LIN {X 0,Y 451.554,Z 691.44,A -85,B 0,C 180,E1 7559.051,E2 7559.051} C_VEL
LIN {X 0,Y 450.796,Z 691.44,A -85,B 0,C 180,E1 7568.723,E2 7568.723} C_VEL
LIN {X 0,Y 450.961,Z 693.251,A -85,B 0,C 180,E1 7574.379,E2 7574.379} C_VEL
LIN {X 0,Y 480.104,Z 749.238,A -85,B 0,C 180,E1 7579.793,E2 7579.793} C_VEL
LIN {X 0,Y 479.486,Z 776.375,A -85,B 0,C 180,E1 7581.127,E2 7581.127} C_VEL
LIN {X 0,Y 471.535,Z 837.542,A -85,B 0,C 180,E1 7585.056,E2 7585.056} C_VEL
LIN {X 0,Y 462.67,Z 892.765,A -85,B 0,C 180,E1 7590.85,E2 7590.85} C_VEL
LIN {X 0,Y 455.796,Z 938.399,A -85,B 0,C 180,E1 7598.248,E2 7598.248} C_VEL
LIN {X 0,Y 452.189,Z 968.248,A -85,B 0,C 180,E1 7605.749,E2 7605.749} C_VEL
LIN {X 0,Y 451.04,Z 986.112,A -85,B 0,C 180,E1 7613.349,E2 7613.349} C_VEL
LIN {X 0,Y 450.564,Z 992.815,A -85,B 0,C 180,E1 7620.766,E2 7620.766} C_VEL
LIN {X 0,Y 451.262,Z 989.016,A -85,B 0,C 180,E1 7628.483,E2 7628.483} C_VEL
LIN {X 0,Y 452.265,Z 972.099,A -85,B 0,C 180,E1 7636.86,E2 7636.86} C_VEL
LIN {X 0,Y 455.576,Z 940.536,A -85,B 0,C 180,E1 7645.223,E2 7645.223} C_VEL
LIN {X 0,Y 462.458,Z 894.509,A -85,B 0,C 180,E1 7652.822,E2 7652.822} C_VEL
LIN {X 0,Y 471.275,Z 839.468,A -85,B 0,C 180,E1 7658.682,E2 7658.682} C_VEL
LIN {X 0,Y 479.234,Z 777.254,A -85,B 0,C 180,E1 7662.749,E2 7662.749} C_VEL
LIN {X 0,Y 480.534,Z 748.867,A -85,B 0,C 180,E1 7664.089,E2 7664.089} C_VEL
LIN {X 0,Y 451.925,Z 695.998,A -85,B 0,C 180,E1 7669.283,E2 7669.283} C_VEL
LIN {X 0,Y 450.465,Z 691.44,A -85,B 0,C 180,E1 7669.758,E2 7669.758} C_VEL
LIN {X 0,Y 450.136,Z 691.44,A -85,B 0,C 180,E1 7679.266,E2 7679.266} C_VEL
LIN {X 0,Y 449.936,Z 691.44,A -85,B 0,C 180,E1 7688.608,E2 7688.608} C_VEL
LIN {X 0,Y 449.949,Z 691.44,A -85,B 0,C 180,E1 7698.876,E2 7698.876} C_VEL
LIN {X 0,Y 450.069,Z 691.44,A -85,B 0,C 180,E1 7709.299,E2 7709.299} C_VEL
LIN {X 0,Y 449.954,Z 691.44,A -85,B 0,C 180,E1 7719.253,E2 7719.253} C_VEL
LIN {X 0,Y 450.985,Z 691.44,A -85,B 0,C 180,E1 7727.357,E2 7727.357} C_VEL
LIN {X 0,Y 450.837,Z 691.44,A -85,B 0,C 180,E1 7737.094,E2 7737.094} C_VEL
LIN {X 0,Y 450.806,Z 691.44,A -85,B 0,C 180,E1 7744.813,E2 7744.813} C_VEL
LIN {X 0,Y 450.666,Z 691.44,A -85,B 0,C 180,E1 7754.61,E2 7754.61} C_VEL
LIN {X 0,Y 450.257,Z 691.44,A -85,B 0,C 180,E1 7764.893,E2 7764.893} C_VEL
LIN {X 0,Y 449.84,Z 691.44,A -85,B 0,C 180,E1 7774.255,E2 7774.255} C_VEL
LIN {X 0,Y 450.159,Z 693.285,A -85,B 0,C 180,E1 7781.816,E2 7781.816} C_VEL
LIN {X 0,Y 483.227,Z 752.373,A -85,B 0,C 180,E1 7787.254,E2 7787.254} C_VEL
LIN {X 0,Y 477.78,Z 816.561,A -85,B 0,C 180,E1 7789.78,E2 7789.78} C_VEL
LIN {X 0,Y 469.391,Z 878.673,A -85,B 0,C 180,E1 7794.175,E2 7794.175} C_VEL
LIN {X 0,Y 468.305,Z 886.117,A -85,B 0,C 180,E1 7794.87,E2 7794.87} C_VEL
LIN {X 0,Y 457.031,Z 913.56,A -85,B 0,C 180,E1 7797.288,E2 7797.288} C_VEL
LIN {X 0,Y 449.955,Z 959.158,A -85,B 0,C 180,E1 7804.083,E2 7804.083} C_VEL
LIN {X 0,Y 445.282,Z 994.231,A -85,B 0,C 180,E1 7812.256,E2 7812.256} C_VEL
LIN {X 0,Y 443.447,Z 1014.285,A -85,B 0,C 180,E1 7820.147,E2 7820.147} C_VEL
LIN {X 0,Y 443.05,Z 1022.147,A -85,B 0,C 180,E1 7827.054,E2 7827.054} C_VEL
LIN {X 0,Y 443.063,Z 1020.767,A -85,B 0,C 180,E1 7834.912,E2 7834.912} C_VEL
LIN {X 0,Y 443.75,Z 1007.555,A -85,B 0,C 180,E1 7843.07,E2 7843.07} C_VEL
LIN {X 0,Y 447.084,Z 979.442,A -85,B 0,C 180,E1 7851.662,E2 7851.662} C_VEL
LIN {X 0,Y 453.089,Z 938.558,A -85,B 0,C 180,E1 7859.353,E2 7859.353} C_VEL
LIN {X 0,Y 461.64,Z 883.668,A -85,B 0,C 180,E1 7865.91,E2 7865.91} C_VEL
LIN {X 0,Y 470.623,Z 820.966,A -85,B 0,C 180,E1 7870.566,E2 7870.566} C_VEL
LIN {X 0,Y 476.046,Z 752.177,A -85,B 0,C 180,E1 7873.483,E2 7873.483} C_VEL
LIN {X 0,Y 441.94,Z 691.44,A -85,B 0,C 180,E1 7879.572,E2 7879.572} C_VEL
LIN {X 0,Y 442.027,Z 691.44,A -85,B 0,C 180,E1 7890.171,E2 7890.171} C_VEL
LIN {X 0,Y 442.1,Z 691.44,A -85,B 0,C 180,E1 7900.989,E2 7900.989} C_VEL
LIN {X 0,Y 442.87,Z 691.44,A -85,B 0,C 180,E1 7911.146,E2 7911.146} C_VEL
LIN {X 0,Y 443.032,Z 691.44,A -85,B 0,C 180,E1 7920.994,E2 7920.994} C_VEL
LIN {X 0,Y 442.705,Z 691.44,A -85,B 0,C 180,E1 7930.877,E2 7930.877} C_VEL
LIN {X 0,Y 442.98,Z 693.318,A -85,B 0,C 180,E1 7933.215,E2 7933.215} C_VEL
LIN {X 0,Y 472.547,Z 748.959,A -85,B 0,C 180,E1 7938.943,E2 7938.943} C_VEL
LIN {X 0,Y 474.866,Z 762.006,A -85,B 0,C 180,E1 7939.835,E2 7939.835} C_VEL
LIN {X 0,Y 466.818,Z 825.923,A -85,B 0,C 180,E1 7943.512,E2 7943.512} C_VEL
LIN {X 0,Y 457.64,Z 882.015,A -85,B 0,C 180,E1 7948.928,E2 7948.928} C_VEL
LIN {X 0,Y 449.947,Z 928.738,A -85,B 0,C 180,E1 7955.962,E2 7955.962} C_VEL
LIN {X 0,Y 445.038,Z 964.744,A -85,B 0,C 180,E1 7964.35,E2 7964.35} C_VEL
LIN {X 0,Y 443.257,Z 984.655,A -85,B 0,C 180,E1 7972.336,E2 7972.336} C_VEL
LIN {X 0,Y 442.582,Z 992.719,A -85,B 0,C 180,E1 7980.186,E2 7980.186} C_VEL
LIN {X 0,Y 443.266,Z 988.627,A -85,B 0,C 180,E1 7988.932,E2 7988.932} C_VEL
LIN {X 0,Y 444.309,Z 970.625,A -85,B 0,C 180,E1 7997.674,E2 7997.674} C_VEL
LIN {X 0,Y 447.986,Z 939.674,A -85,B 0,C 180,E1 8005.832,E2 8005.832} C_VEL
LIN {X 0,Y 455.506,Z 893.468,A -85,B 0,C 180,E1 8013.528,E2 8013.528} C_VEL
LIN {X 0,Y 464.916,Z 838.34,A -85,B 0,C 180,E1 8019.394,E2 8019.394} C_VEL
LIN {X 0,Y 473.409,Z 775.784,A -85,B 0,C 180,E1 8023.457,E2 8023.457} C_VEL
LIN {X 0,Y 474.106,Z 751.685,A -85,B 0,C 180,E1 8024.661,E2 8024.661} C_VEL
LIN {X 0,Y 445.382,Z 697.645,A -85,B 0,C 180,E1 8030.143,E2 8030.143} C_VEL
LIN {X 0,Y 442.399,Z 691.44,A -85,B 0,C 180,E1 8031.112,E2 8031.112} C_VEL
LIN {X 0,Y 442.119,Z 691.44,A -85,B 0,C 180,E1 8039.85,E2 8039.85} C_VEL
LIN {X 0,Y 441.891,Z 691.44,A -85,B 0,C 180,E1 8049.446,E2 8049.446} C_VEL
LIN {X 0,Y 441.873,Z 691.44,A -85,B 0,C 180,E1 8057.955,E2 8057.955} C_VEL
LIN {X 0,Y 441.946,Z 691.44,A -85,B 0,C 180,E1 8067.839,E2 8067.839} C_VEL
LIN {X 0,Y 441.935,Z 691.44,A -85,B 0,C 180,E1 8076.734,E2 8076.734} C_VEL
LIN {X 0,Y 442.969,Z 691.44,A -85,B 0,C 180,E1 8087.528,E2 8087.528} C_VEL
LIN {X 0,Y 442.866,Z 691.44,A -85,B 0,C 180,E1 8097.041,E2 8097.041} C_VEL
LIN {X 0,Y 442.821,Z 691.44,A -85,B 0,C 180,E1 8104.9,E2 8104.9} C_VEL
LIN {X 0,Y 442.657,Z 691.44,A -85,B 0,C 180,E1 8114.88,E2 8114.88} C_VEL
LIN {X 0,Y 442.205,Z 691.44,A -85,B 0,C 180,E1 8125.379,E2 8125.379} C_VEL
LIN {X 0,Y 441.848,Z 691.44,A -85,B 0,C 180,E1 8136.182,E2 8136.182} C_VEL
LIN {X 0,Y 442.043,Z 692.748,A -85,B 0,C 180,E1 8140.669,E2 8140.669} C_VEL
LIN {X 0,Y 477.063,Z 755.273,A -85,B 0,C 180,E1 8146.678,E2 8146.678} C_VEL
LIN {X 0,Y 471.042,Z 819.946,A -85,B 0,C 180,E1 8149.353,E2 8149.353} C_VEL
LIN {X 0,Y 462.246,Z 881.197,A -85,B 0,C 180,E1 8153.834,E2 8153.834} C_VEL
LIN {X 0,Y 457.031,Z 913.56,A -85,B 0,C 180,E1 8157.288,E2 8157.288} C_VEL
LIN {X 0,Y 445.432,Z 938.523,A -85,B 0,C 180,E1 8160.14,E2 8160.14} C_VEL
LIN {X 0,Y 438.964,Z 978.353,A -85,B 0,C 180,E1 8167.648,E2 8167.648} C_VEL
LIN {X 0,Y 435.816,Z 1004.336,A -85,B 0,C 180,E1 8175.377,E2 8175.377} C_VEL
LIN {X 0,Y 435.092,Z 1019.244,A -85,B 0,C 180,E1 8183.454,E2 8183.454} C_VEL
LIN {X 0,Y 435.342,Z 1022.837,A -85,B 0,C 180,E1 8190.998,E2 8190.998} C_VEL
LIN {X 0,Y 435.357,Z 1015.886,A -85,B 0,C 180,E1 8199.024,E2 8199.024} C_VEL
LIN {X 0,Y 436.862,Z 995.719,A -85,B 0,C 180,E1 8207.643,E2 8207.643} C_VEL
LIN {X 0,Y 441.422,Z 962.929,A -85,B 0,C 180,E1 8215.664,E2 8215.664} C_VEL
LIN {X 0,Y 449.432,Z 915.459,A -85,B 0,C 180,E1 8222.997,E2 8222.997} C_VEL
LIN {X 0,Y 459.298,Z 857.062,A -85,B 0,C 180,E1 8228.768,E2 8228.768} C_VEL
LIN {X 0,Y 467.582,Z 794.293,A -85,B 0,C 180,E1 8232.533,E2 8232.533} C_VEL
LIN {X 0,Y 469.791,Z 755.185,A -85,B 0,C 180,E1 8234.086,E2 8234.086} C_VEL
LIN {X 0,Y 436.487,Z 697.36,A -85,B 0,C 180,E1 8240.149,E2 8240.149} C_VEL
LIN {X 0,Y 433.802,Z 691.44,A -85,B 0,C 180,E1 8240.877,E2 8240.877} C_VEL
LIN {X 0,Y 434.008,Z 691.44,A -85,B 0,C 180,E1 8251.859,E2 8251.859} C_VEL
LIN {X 0,Y 434.256,Z 691.44,A -85,B 0,C 180,E1 8262.74,E2 8262.74} C_VEL
LIN {X 0,Y 434.924,Z 691.44,A -85,B 0,C 180,E1 8273.001,E2 8273.001} C_VEL
LIN {X 0,Y 435.026,Z 691.44,A -85,B 0,C 180,E1 8281.013,E2 8281.013} C_VEL
LIN {X 0,Y 434.694,Z 691.44,A -85,B 0,C 180,E1 8291.08,E2 8291.08} C_VEL
LIN {X 0,Y 435.021,Z 693.636,A -85,B 0,C 180,E1 8291.977,E2 8291.977} C_VEL
LIN {X 0,Y 464.673,Z 747.641,A -85,B 0,C 180,E1 8297.959,E2 8297.959} C_VEL
LIN {X 0,Y 468.849,Z 762.644,A -85,B 0,C 180,E1 8299.199,E2 8299.199} C_VEL
LIN {X 0,Y 460.363,Z 826.705,A -85,B 0,C 180,E1 8302.927,E2 8302.927} C_VEL
LIN {X 0,Y 450.621,Z 882.973,A -85,B 0,C 180,E1 8308.447,E2 8308.447} C_VEL
LIN {X 0,Y 442.51,Z 928.888,A -85,B 0,C 180,E1 8315.491,E2 8315.491} C_VEL
LIN {X 0,Y 437.286,Z 964.581,A -85,B 0,C 180,E1 8323.978,E2 8323.978} C_VEL
LIN {X 0,Y 435.243,Z 985.065,A -85,B 0,C 180,E1 8332.398,E2 8332.398} C_VEL
LIN {X 0,Y 434.561,Z 992.463,A -85,B 0,C 180,E1 8339.578,E2 8339.578} C_VEL
LIN {X 0,Y 435.121,Z 990.295,A -85,B 0,C 180,E1 8347.542,E2 8347.542} C_VEL
LIN {X 0,Y 436.37,Z 974.559,A -85,B 0,C 180,E1 8356.49,E2 8356.49} C_VEL
LIN {X 0,Y 439.717,Z 945.125,A -85,B 0,C 180,E1 8365.051,E2 8365.051} C_VEL
LIN {X 0,Y 447.115,Z 901.895,A -85,B 0,C 180,E1 8372.919,E2 8372.919} C_VEL
LIN {X 0,Y 456.677,Z 848.952,A -85,B 0,C 180,E1 8379.082,E2 8379.082} C_VEL
LIN {X 0,Y 465.74,Z 787.5,A -85,B 0,C 180,E1 8383.545,E2 8383.545} C_VEL
LIN {X 0,Y 468.049,Z 755.229,A -85,B 0,C 180,E1 8385.176,E2 8385.176} C_VEL
LIN {X 0,Y 440.965,Z 703.44,A -85,B 0,C 180,E1 8390.624,E2 8390.624} C_VEL
LIN {X 0,Y 434.298,Z 691.44,A -85,B 0,C 180,E1 8392.194,E2 8392.194} C_VEL
LIN {X 0,Y 433.924,Z 691.44,A -85,B 0,C 180,E1 8402.827,E2 8402.827} C_VEL
LIN {X 0,Y 433.83,Z 691.44,A -85,B 0,C 180,E1 8413.011,E2 8413.011} C_VEL
LIN {X 0,Y 433.75,Z 691.44,A -85,B 0,C 180,E1 8422.244,E2 8422.244} C_VEL
LIN {X 0,Y 434.015,Z 691.44,A -85,B 0,C 180,E1 8433.081,E2 8433.081} C_VEL
LIN {X 0,Y 434.843,Z 691.44,A -85,B 0,C 180,E1 8444.818,E2 8444.818} C_VEL
LIN {X 0,Y 435.01,Z 691.44,A -85,B 0,C 180,E1 8454.985,E2 8454.985} C_VEL
LIN {X 0,Y 435.081,Z 691.44,A -85,B 0,C 180,E1 8462.984,E2 8462.984} C_VEL
LIN {X 0,Y 434.639,Z 691.44,A -85,B 0,C 180,E1 8473.099,E2 8473.099} C_VEL
LIN {X 0,Y 434.257,Z 691.44,A -85,B 0,C 180,E1 8483.672,E2 8483.672} C_VEL
LIN {X 0,Y 433.815,Z 691.44,A -85,B 0,C 180,E1 8494.705,E2 8494.705} C_VEL
LIN {X 0,Y 433.956,Z 692.746,A -85,B 0,C 180,E1 8499.468,E2 8499.468} C_VEL
LIN {X 0,Y 469.825,Z 755.777,A -85,B 0,C 180,E1 8505.884,E2 8505.884} C_VEL
LIN {X 0,Y 464.026,Z 825.724,A -85,B 0,C 180,E1 8509.052,E2 8509.052} C_VEL
LIN {X 0,Y 454.868,Z 884.496,A -85,B 0,C 180,E1 8513.572,E2 8513.572} C_VEL
LIN {X 0,Y 445.432,Z 938.523,A -85,B 0,C 180,E1 8520.14,E2 8520.14} C_VEL
LIN {X 0,Y 434.61,Z 960.552,A -85,B 0,C 180,E1 8523.479,E2 8523.479} C_VEL
LIN {X 0,Y 429.713,Z 993.824,A -85,B 0,C 180,E1 8531.467,E2 8531.467} C_VEL
LIN {X 0,Y 427.573,Z 1014.285,A -85,B 0,C 180,E1 8539.777,E2 8539.777} C_VEL
LIN {X 0,Y 427.056,Z 1022.147,A -85,B 0,C 180,E1 8546.944,E2 8546.944} C_VEL
LIN {X 0,Y 427.087,Z 1020.766,A -85,B 0,C 180,E1 8555.096,E2 8555.096} C_VEL
LIN {X 0,Y 428.068,Z 1006.921,A -85,B 0,C 180,E1 8563.845,E2 8563.845} C_VEL
LIN {X 0,Y 431.896,Z 978.302,A -85,B 0,C 180,E1 8572.737,E2 8572.737} C_VEL
LIN {X 0,Y 438.853,Z 936.044,A -85,B 0,C 180,E1 8580.668,E2 8580.668} C_VEL
LIN {X 0,Y 448.501,Z 881.198,A -85,B 0,C 180,E1 8587.31,E2 8587.31} C_VEL
LIN {X 0,Y 458.407,Z 817.94,A -85,B 0,C 180,E1 8592.02,E2 8592.02} C_VEL
LIN {X 0,Y 463.715,Z 758.59,A -85,B 0,C 180,E1 8594.657,E2 8594.657} C_VEL
LIN {X 0,Y 432.524,Z 703.466,A -85,B 0,C 180,E1 8600.626,E2 8600.626} C_VEL
LIN {X 0,Y 425.74,Z 691.44,A -85,B 0,C 180,E1 8602.433,E2 8602.433} C_VEL
LIN {X 0,Y 425.979,Z 691.44,A -85,B 0,C 180,E1 8613.582,E2 8613.582} C_VEL
LIN {X 0,Y 426.337,Z 691.44,A -85,B 0,C 180,E1 8624.536,E2 8624.536} C_VEL
LIN {X 0,Y 426.827,Z 691.44,A -85,B 0,C 180,E1 8634.916,E2 8634.916} C_VEL
LIN {X 0,Y 426.878,Z 691.44,A -85,B 0,C 180,E1 8643.07,E2 8643.07} C_VEL
LIN {X 0,Y 426.829,Z 693.053,A -85,B 0,C 180,E1 8650.574,E2 8650.574} C_VEL
LIN {X 0,Y 456.913,Z 746.746,A -85,B 0,C 180,E1 8656.957,E2 8656.957} C_VEL
LIN {X 0,Y 462.493,Z 766.687,A -85,B 0,C 180,E1 8658.693,E2 8658.693} C_VEL
LIN {X 0,Y 453.603,Z 829.727,A -85,B 0,C 180,E1 8662.495,E2 8662.495} C_VEL
LIN {X 0,Y 443.125,Z 886.449,A -85,B 0,C 180,E1 8668.262,E2 8668.262} C_VEL
LIN {X 0,Y 434.551,Z 932.151,A -85,B 0,C 180,E1 8675.584,E2 8675.584} C_VEL
LIN {X 0,Y 428.946,Z 967.211,A -85,B 0,C 180,E1 8684.489,E2 8684.489} C_VEL
LIN {X 0,Y 427.137,Z 986.415,A -85,B 0,C 180,E1 8693.07,E2 8693.07} C_VEL
LIN {X 0,Y 426.463,Z 992.905,A -85,B 0,C 180,E1 8701.289,E2 8701.289} C_VEL
LIN {X 0,Y 427.2,Z 988.636,A -85,B 0,C 180,E1 8709.193,E2 8709.193} C_VEL
LIN {X 0,Y 428.407,Z 971.752,A -85,B 0,C 180,E1 8717.843,E2 8717.843} C_VEL
LIN {X 0,Y 432.819,Z 939.838,A -85,B 0,C 180,E1 8726.734,E2 8726.734} C_VEL
LIN {X 0,Y 441.104,Z 895.84,A -85,B 0,C 180,E1 8734.382,E2 8734.382} C_VEL
LIN {X 0,Y 451.537,Z 841.543,A -85,B 0,C 180,E1 8740.408,E2 8740.408} C_VEL
LIN {X 0,Y 461.059,Z 778.462,A -85,B 0,C 180,E1 8744.659,E2 8744.659} C_VEL
LIN {X 0,Y 461.808,Z 758.295,A -85,B 0,C 180,E1 8745.753,E2 8745.753} C_VEL
LIN {X 0,Y 436.098,Z 708.579,A -85,B 0,C 180,E1 8751.184,E2 8751.184} C_VEL
LIN {X 0,Y 426.272,Z 691.44,A -85,B 0,C 180,E1 8753.157,E2 8753.157} C_VEL
LIN {X 0,Y 425.866,Z 691.44,A -85,B 0,C 180,E1 8763.529,E2 8763.529} C_VEL
LIN {X 0,Y 425.806,Z 691.44,A -85,B 0,C 180,E1 8774.027,E2 8774.027} C_VEL
LIN {X 0,Y 425.748,Z 691.44,A -85,B 0,C 180,E1 8783.972,E2 8783.972} C_VEL
LIN {X 0,Y 426.016,Z 691.44,A -85,B 0,C 180,E1 8793.553,E2 8793.553} C_VEL
LIN {X 0,Y 426.78,Z 691.44,A -85,B 0,C 180,E1 8804.524,E2 8804.524} C_VEL
LIN {X 0,Y 427.001,Z 691.44,A -85,B 0,C 180,E1 8814.89,E2 8814.89} C_VEL
LIN {X 0,Y 427.065,Z 691.44,A -85,B 0,C 180,E1 8823.041,E2 8823.041} C_VEL
LIN {X 0,Y 426.619,Z 691.44,A -85,B 0,C 180,E1 8833.35,E2 8833.35} C_VEL
LIN {X 0,Y 426.172,Z 691.44,A -85,B 0,C 180,E1 8844.15,E2 8844.15} C_VEL
LIN {X 0,Y 425.796,Z 691.44,A -85,B 0,C 180,E1 8853.504,E2 8853.504} C_VEL
LIN {X 0,Y 425.926,Z 693.215,A -85,B 0,C 180,E1 8858.227,E2 8858.227} C_VEL
LIN {X 0,Y 461.569,Z 754.086,A -85,B 0,C 180,E1 8864.861,E2 8864.861} C_VEL
LIN {X 0,Y 464.491,Z 766.283,A -85,B 0,C 180,E1 8865.689,E2 8865.689} C_VEL
LIN {X 0,Y 456.915,Z 831.706,A -85,B 0,C 180,E1 8868.774,E2 8868.774} C_VEL
LIN {X 0,Y 446.908,Z 891.589,A -85,B 0,C 180,E1 8873.698,E2 8873.698} C_VEL
LIN {X 0,Y 437.196,Z 943.334,A -85,B 0,C 180,E1 8880.424,E2 8880.424} C_VEL
LIN {X 0,Y 434.61,Z 960.552,A -85,B 0,C 180,E1 8883.479,E2 8883.479} C_VEL
LIN {X 0,Y 423.366,Z 979.613,A -85,B 0,C 180,E1 8887.193,E2 8887.193} C_VEL
LIN {X 0,Y 419.891,Z 1005.675,A -85,B 0,C 180,E1 8895.345,E2 8895.345} C_VEL
LIN {X 0,Y 419.067,Z 1018.682,A -85,B 0,C 180,E1 8902.718,E2 8902.718} C_VEL
LIN {X 0,Y 419.337,Z 1022.836,A -85,B 0,C 180,E1 8911.036,E2 8911.036} C_VEL
LIN {X 0,Y 419.336,Z 1015.886,A -85,B 0,C 180,E1 8919.372,E2 8919.372} C_VEL
LIN {X 0,Y 420.99,Z 997.104,A -85,B 0,C 180,E1 8927.843,E2 8927.843} C_VEL
LIN {X 0,Y 425.962,Z 964.688,A -85,B 0,C 180,E1 8936.132,E2 8936.132} C_VEL
LIN {X 0,Y 434.995,Z 916.695,A -85,B 0,C 180,E1 8943.931,E2 8943.931} C_VEL
LIN {X 0,Y 446.071,Z 858.144,A -85,B 0,C 180,E1 8949.93,E2 8949.93} C_VEL
LIN {X 0,Y 455.377,Z 795.802,A -85,B 0,C 180,E1 8953.801,E2 8953.801} C_VEL
LIN {X 0,Y 457.53,Z 761.525,A -85,B 0,C 180,E1 8955.277,E2 8955.277} C_VEL
LIN {X 0,Y 428.214,Z 708.933,A -85,B 0,C 180,E1 8961.2,E2 8961.2} C_VEL
LIN {X 0,Y 417.729,Z 691.44,A -85,B 0,C 180,E1 8963.636,E2 8963.636} C_VEL
LIN {X 0,Y 417.903,Z 691.44,A -85,B 0,C 180,E1 8973.03,E2 8973.03} C_VEL
LIN {X 0,Y 418.277,Z 691.44,A -85,B 0,C 180,E1 8984.23,E2 8984.23} C_VEL
LIN {X 0,Y 418.828,Z 691.44,A -85,B 0,C 180,E1 8995.16,E2 8995.16} C_VEL
LIN {X 0,Y 418.875,Z 691.44,A -85,B 0,C 180,E1 9003.128,E2 9003.128} C_VEL
LIN {X 0,Y 418.957,Z 693.291,A -85,B 0,C 180,E1 9009.129,E2 9009.129} C_VEL
LIN {X 0,Y 447.481,Z 742.324,A -85,B 0,C 180,E1 9015.519,E2 9015.519} C_VEL
LIN {X 0,Y 456.404,Z 769.016,A -85,B 0,C 180,E1 9018.099,E2 9018.099} C_VEL
LIN {X 0,Y 447.195,Z 830.655,A -85,B 0,C 180,E1 9021.892,E2 9021.892} C_VEL
LIN {X 0,Y 436.217,Z 887.146,A -85,B 0,C 180,E1 9027.722,E2 9027.722} C_VEL
LIN {X 0,Y 427.316,Z 931.762,A -85,B 0,C 180,E1 9034.962,E2 9034.962} C_VEL
LIN {X 0,Y 421.506,Z 965.772,A -85,B 0,C 180,E1 9043.661,E2 9043.661} C_VEL
LIN {X 0,Y 419.279,Z 985.435,A -85,B 0,C 180,E1 9052.258,E2 9052.258} C_VEL
LIN {X 0,Y 418.483,Z 992.818,A -85,B 0,C 180,E1 9060.688,E2 9060.688} C_VEL
LIN {X 0,Y 419.2,Z 989.225,A -85,B 0,C 180,E1 9068.776,E2 9068.776} C_VEL
LIN {X 0,Y 420.446,Z 972.894,A -85,B 0,C 180,E1 9077.704,E2 9077.704} C_VEL
LIN {X 0,Y 424.898,Z 942.401,A -85,B 0,C 180,E1 9086.673,E2 9086.673} C_VEL
LIN {X 0,Y 433.661,Z 898.569,A -85,B 0,C 180,E1 9094.612,E2 9094.612} C_VEL
LIN {X 0,Y 444.87,Z 843.076,A -85,B 0,C 180,E1 9100.939,E2 9100.939} C_VEL
LIN {X 0,Y 454.776,Z 780.809,A -85,B 0,C 180,E1 9105.236,E2 9105.236} C_VEL
LIN {X 0,Y 455.561,Z 761.257,A -85,B 0,C 180,E1 9106.35,E2 9106.35} C_VEL
LIN {X 0,Y 429.428,Z 710.166,A -85,B 0,C 180,E1 9112.142,E2 9112.142} C_VEL
LIN {X 0,Y 418.215,Z 691.44,A -85,B 0,C 180,E1 9114.665,E2 9114.665} C_VEL
LIN {X 0,Y 417.701,Z 691.44,A -85,B 0,C 180,E1 9125.172,E2 9125.172} C_VEL
LIN {X 0,Y 417.747,Z 691.44,A -85,B 0,C 180,E1 9135.105,E2 9135.105} C_VEL
LIN {X 0,Y 417.746,Z 691.44,A -85,B 0,C 180,E1 9145.727,E2 9145.727} C_VEL
LIN {X 0,Y 417.943,Z 691.44,A -85,B 0,C 180,E1 9155.312,E2 9155.312} C_VEL
LIN {X 0,Y 418.876,Z 691.44,A -85,B 0,C 180,E1 9166.37,E2 9166.37} C_VEL
LIN {X 0,Y 418.869,Z 691.44,A -85,B 0,C 180,E1 9176.872,E2 9176.872} C_VEL
LIN {X 0,Y 418.832,Z 691.44,A -85,B 0,C 180,E1 9185.181,E2 9185.181} C_VEL
LIN {X 0,Y 418.489,Z 691.44,A -85,B 0,C 180,E1 9196.056,E2 9196.056} C_VEL
LIN {X 0,Y 418,Z 691.44,A -85,B 0,C 180,E1 9207.189,E2 9207.189} C_VEL
LIN {X 0,Y 417.818,Z 692.822,A -85,B 0,C 180,E1 9216.873,E2 9216.873} C_VEL
LIN {X 0,Y 454.81,Z 755.444,A -85,B 0,C 180,E1 9224.079,E2 9224.079} C_VEL
LIN {X 0,Y 458.441,Z 768.769,A -85,B 0,C 180,E1 9225.079,E2 9225.079} C_VEL
LIN {X 0,Y 450.44,Z 833.237,A -85,B 0,C 180,E1 9228.216,E2 9228.216} C_VEL
LIN {X 0,Y 439.853,Z 893.141,A -85,B 0,C 180,E1 9233.253,E2 9233.253} C_VEL
LIN {X 0,Y 429.326,Z 946.123,A -85,B 0,C 180,E1 9240.387,E2 9240.387} C_VEL
LIN {X 0,Y 423.366,Z 979.613,A -85,B 0,C 180,E1 9247.193,E2 9247.193} C_VEL
LIN {X 0,Y 413.778,Z 995.457,A -85,B 0,C 180,E1 9251.347,E2 9251.347} C_VEL
LIN {X 0,Y 411.346,Z 1015.885,A -85,B 0,C 180,E1 9260.443,E2 9260.443} C_VEL
LIN {X 0,Y 410.914,Z 1022.836,A -85,B 0,C 180,E1 9268.941,E2 9268.941} C_VEL
LIN {X 0,Y 411.395,Z 1018.684,A -85,B 0,C 180,E1 9277.418,E2 9277.418} C_VEL
LIN {X 0,Y 412.834,Z 1001.069,A -85,B 0,C 180,E1 9286.72,E2 9286.72} C_VEL
LIN {X 0,Y 417.568,Z 969.238,A -85,B 0,C 180,E1 9295.567,E2 9295.567} C_VEL
LIN {X 0,Y 426.454,Z 924.125,A -85,B 0,C 180,E1 9303.475,E2 9303.475} C_VEL
LIN {X 0,Y 437.846,Z 868.131,A -85,B 0,C 180,E1 9309.742,E2 9309.742} C_VEL
LIN {X 0,Y 448.239,Z 804.001,A -85,B 0,C 180,E1 9314.113,E2 9314.113} C_VEL
LIN {X 0,Y 451.602,Z 764.858,A -85,B 0,C 180,E1 9315.874,E2 9315.874} C_VEL
LIN {X 0,Y 423.26,Z 713.124,A -85,B 0,C 180,E1 9321.942,E2 9321.942} C_VEL
LIN {X 0,Y 409.701,Z 691.44,A -85,B 0,C 180,E1 9325.382,E2 9325.382} C_VEL
LIN {X 0,Y 409.891,Z 691.44,A -85,B 0,C 180,E1 9335.106,E2 9335.106} C_VEL
LIN {X 0,Y 410.281,Z 691.44,A -85,B 0,C 180,E1 9346.108,E2 9346.108} C_VEL
LIN {X 0,Y 411.043,Z 691.44,A -85,B 0,C 180,E1 9356.841,E2 9356.841} C_VEL
LIN {X 0,Y 411.202,Z 693.44,A -85,B 0,C 180,E1 9367.567,E2 9367.567} C_VEL
LIN {X 0,Y 439.184,Z 740.651,A -85,B 0,C 180,E1 9374.262,E2 9374.262} C_VEL
LIN {X 0,Y 450.431,Z 770.964,A -85,B 0,C 180,E1 9377.47,E2 9377.47} C_VEL
LIN {X 0,Y 440.671,Z 832.485,A -85,B 0,C 180,E1 9381.346,E2 9381.346} C_VEL
LIN {X 0,Y 428.947,Z 889.607,A -85,B 0,C 180,E1 9387.387,E2 9387.387} C_VEL
LIN {X 0,Y 419.206,Z 935.498,A -85,B 0,C 180,E1 9395.17,E2 9395.17} C_VEL
LIN {X 0,Y 413.14,Z 968.742,A -85,B 0,C 180,E1 9404.251,E2 9404.251} C_VEL
LIN {X 0,Y 411.244,Z 986.116,A -85,B 0,C 180,E1 9412.502,E2 9412.502} C_VEL
LIN {X 0,Y 410.469,Z 992.767,A -85,B 0,C 180,E1 9420.318,E2 9420.318} C_VEL
LIN {X 0,Y 411.215,Z 988.641,A -85,B 0,C 180,E1 9429.477,E2 9429.477} C_VEL
LIN {X 0,Y 412.553,Z 972.268,A -85,B 0,C 180,E1 9438.328,E2 9438.328} C_VEL
LIN {X 0,Y 417.445,Z 942.392,A -85,B 0,C 180,E1 9447.202,E2 9447.202} C_VEL
LIN {X 0,Y 426.809,Z 898.383,A -85,B 0,C 180,E1 9455.265,E2 9455.265} C_VEL
LIN {X 0,Y 438.505,Z 843.291,A -85,B 0,C 180,E1 9461.605,E2 9461.605} C_VEL
LIN {X 0,Y 448.789,Z 781.728,A -85,B 0,C 180,E1 9465.897,E2 9465.897} C_VEL
LIN {X 0,Y 449.492,Z 764.735,A -85,B 0,C 180,E1 9466.896,E2 9466.896} C_VEL
LIN {X 0,Y 424.732,Z 715.504,A -85,B 0,C 180,E1 9472.711,E2 9472.711} C_VEL
LIN {X 0,Y 410.066,Z 691.44,A -85,B 0,C 180,E1 9476.16,E2 9476.16} C_VEL
LIN {X 0,Y 409.721,Z 691.44,A -85,B 0,C 180,E1 9487.674,E2 9487.674} C_VEL
LIN {X 0,Y 409.668,Z 691.44,A -85,B 0,C 180,E1 9496.738,E2 9496.738} C_VEL
LIN {X 0,Y 409.745,Z 691.44,A -85,B 0,C 180,E1 9507.513,E2 9507.513} C_VEL
LIN {X 0,Y 409.849,Z 691.44,A -85,B 0,C 180,E1 9517.113,E2 9517.113} C_VEL
LIN {X 0,Y 410.849,Z 691.44,A -85,B 0,C 180,E1 9526.098,E2 9526.098} C_VEL
LIN {X 0,Y 410.887,Z 691.44,A -85,B 0,C 180,E1 9536.811,E2 9536.811} C_VEL
LIN {X 0,Y 410.823,Z 691.44,A -85,B 0,C 180,E1 9545.282,E2 9545.282} C_VEL
LIN {X 0,Y 410.494,Z 691.44,A -85,B 0,C 180,E1 9556.077,E2 9556.077} C_VEL
LIN {X 0,Y 409.954,Z 691.44,A -85,B 0,C 180,E1 9567.537,E2 9567.537} C_VEL
LIN {X 0,Y 409.803,Z 693,A -85,B 0,C 180,E1 9575.462,E2 9575.462} C_VEL
LIN {X 0,Y 446.54,Z 753.897,A -85,B 0,C 180,E1 9582.966,E2 9582.966} C_VEL
LIN {X 0,Y 452.372,Z 771.841,A -85,B 0,C 180,E1 9584.48,E2 9584.48} C_VEL
LIN {X 0,Y 443.58,Z 837.386,A -85,B 0,C 180,E1 9587.816,E2 9587.816} C_VEL
LIN {X 0,Y 432.628,Z 895.645,A -85,B 0,C 180,E1 9592.921,E2 9592.921} C_VEL
LIN {X 0,Y 421.736,Z 947.525,A -85,B 0,C 180,E1 9600.12,E2 9600.12} C_VEL
LIN {X 0,Y 414.671,Z 986.437,A -85,B 0,C 180,E1 9608.642,E2 9608.642} C_VEL
LIN {X 0,Y 413.778,Z 995.457,A -85,B 0,C 180,E1 9611.347,E2 9611.347} C_VEL
LIN {X 0,Y 403.834,Z 1007.667,A -85,B 0,C 180,E1 9615.812,E2 9615.812} C_VEL
LIN {X 0,Y 403.301,Z 1020.764,A -85,B 0,C 180,E1 9624.602,E2 9624.602} C_VEL
LIN {X 0,Y 403.189,Z 1022.147,A -85,B 0,C 180,E1 9633.236,E2 9633.236} C_VEL
LIN {X 0,Y 403.424,Z 1012.166,A -85,B 0,C 180,E1 9641.94,E2 9641.94} C_VEL
LIN {X 0,Y 406.41,Z 989.492,A -85,B 0,C 180,E1 9650.777,E2 9650.777} C_VEL
LIN {X 0,Y 413.722,Z 950.985,A -85,B 0,C 180,E1 9659.682,E2 9659.682} C_VEL
LIN {X 0,Y 424.292,Z 901.616,A -85,B 0,C 180,E1 9666.966,E2 9666.966} C_VEL
LIN {X 0,Y 436.418,Z 841.519,A -85,B 0,C 180,E1 9672.538,E2 9672.538} C_VEL
LIN {X 0,Y 445.892,Z 778.77,A -85,B 0,C 180,E1 9675.918,E2 9675.918} C_VEL
LIN {X 0,Y 445.041,Z 766.744,A -85,B 0,C 180,E1 9676.645,E2 9676.645} C_VEL
LIN {X 0,Y 418.043,Z 716.91,A -85,B 0,C 180,E1 9682.789,E2 9682.789} C_VEL
LIN {X 0,Y 401.709,Z 691.44,A -85,B 0,C 180,E1 9687.565,E2 9687.565} C_VEL
LIN {X 0,Y 401.796,Z 691.44,A -85,B 0,C 180,E1 9697.723,E2 9697.723} C_VEL
LIN {X 0,Y 402.393,Z 691.44,A -85,B 0,C 180,E1 9708.048,E2 9708.048} C_VEL
LIN {X 0,Y 403.477,Z 691.44,A -85,B 0,C 180,E1 9718.937,E2 9718.937} C_VEL
LIN {X 0,Y 403.194,Z 693.298,A -85,B 0,C 180,E1 9725.762,E2 9725.762} C_VEL
LIN {X 0,Y 430.869,Z 738.634,A -85,B 0,C 180,E1 9732.888,E2 9732.888} C_VEL
LIN {X 0,Y 444.338,Z 774.258,A -85,B 0,C 180,E1 9736.884,E2 9736.884} C_VEL
LIN {X 0,Y 433.824,Z 836.126,A -85,B 0,C 180,E1 9740.937,E2 9740.937} C_VEL
LIN {X 0,Y 421.784,Z 891.464,A -85,B 0,C 180,E1 9746.976,E2 9746.976} C_VEL
LIN {X 0,Y 411.633,Z 936.726,A -85,B 0,C 180,E1 9754.854,E2 9754.854} C_VEL
LIN {X 0,Y 405.457,Z 968.827,A -85,B 0,C 180,E1 9763.824,E2 9763.824} C_VEL
LIN {X 0,Y 403.188,Z 986.968,A -85,B 0,C 180,E1 9772.896,E2 9772.896} C_VEL
LIN {X 0,Y 402.4,Z 992.995,A -85,B 0,C 180,E1 9781.874,E2 9781.874} C_VEL
LIN {X 0,Y 403.206,Z 988.464,A -85,B 0,C 180,E1 9789.815,E2 9789.815} C_VEL
LIN {X 0,Y 404.684,Z 972.572,A -85,B 0,C 180,E1 9798.646,E2 9798.646} C_VEL
LIN {X 0,Y 409.803,Z 943.52,A -85,B 0,C 180,E1 9807.484,E2 9807.484} C_VEL
LIN {X 0,Y 419.617,Z 899.967,A -85,B 0,C 180,E1 9815.687,E2 9815.687} C_VEL
LIN {X 0,Y 431.935,Z 844.772,A -85,B 0,C 180,E1 9822.17,E2 9822.17} C_VEL
LIN {X 0,Y 442.79,Z 783.041,A -85,B 0,C 180,E1 9826.553,E2 9826.553} C_VEL
LIN {X 0,Y 443.377,Z 767.856,A -85,B 0,C 180,E1 9827.488,E2 9827.488} C_VEL
LIN {X 0,Y 419.067,Z 719.123,A -85,B 0,C 180,E1 9833.507,E2 9833.507} C_VEL
LIN {X 0,Y 402.028,Z 691.44,A -85,B 0,C 180,E1 9837.498,E2 9837.498} C_VEL
LIN {X 0,Y 401.603,Z 691.44,A -85,B 0,C 180,E1 9848.573,E2 9848.573} C_VEL
LIN {X 0,Y 401.573,Z 691.44,A -85,B 0,C 180,E1 9858.596,E2 9858.596} C_VEL
LIN {X 0,Y 401.753,Z 691.44,A -85,B 0,C 180,E1 9869.334,E2 9869.334} C_VEL
LIN {X 0,Y 401.862,Z 691.44,A -85,B 0,C 180,E1 9878.968,E2 9878.968} C_VEL
LIN {X 0,Y 402.794,Z 691.44,A -85,B 0,C 180,E1 9888.03,E2 9888.03} C_VEL
LIN {X 0,Y 403.037,Z 691.44,A -85,B 0,C 180,E1 9898.941,E2 9898.941} C_VEL
LIN {X 0,Y 402.775,Z 691.44,A -85,B 0,C 180,E1 9909.743,E2 9909.743} C_VEL
LIN {X 0,Y 402.2,Z 691.44,A -85,B 0,C 180,E1 9920.982,E2 9920.982} C_VEL
LIN {X 0,Y 401.671,Z 691.44,A -85,B 0,C 180,E1 9931.777,E2 9931.777} C_VEL
LIN {X 0,Y 401.903,Z 693.42,A -85,B 0,C 180,E1 9933.998,E2 9933.998} C_VEL
LIN {X 0,Y 437.811,Z 751.555,A -85,B 0,C 180,E1 9941.699,E2 9941.699} C_VEL
LIN {X 0,Y 446.347,Z 774.056,A -85,B 0,C 180,E1 9943.842,E2 9943.842} C_VEL
LIN {X 0,Y 436.813,Z 840.842,A -85,B 0,C 180,E1 9947.353,E2 9947.353} C_VEL
LIN {X 0,Y 424.944,Z 899.951,A -85,B 0,C 180,E1 9952.78,E2 9952.78} C_VEL
LIN {X 0,Y 413.899,Z 949.824,A -85,B 0,C 180,E1 9960.031,E2 9960.031} C_VEL
LIN {X 0,Y 406.61,Z 988.375,A -85,B 0,C 180,E1 9968.847,E2 9968.847} C_VEL
LIN {X 0,Y 403.834,Z 1007.667,A -85,B 0,C 180,E1 9975.812,E2 9975.812} C_VEL
LIN {X 0,Y 395.304,Z 1016.34,A -85,B 0,C 180,E1 9980.625,E2 9980.625} C_VEL
LIN {X 0,Y 394.932,Z 1022.664,A -85,B 0,C 180,E1 9988.899,E2 9988.899} C_VEL
LIN {X 0,Y 395.422,Z 1018.387,A -85,B 0,C 180,E1 9997.719,E2 9997.719} C_VEL
LIN {X 0,Y 396.951,Z 1001.075,A -85,B 0,C 180,E1 10007.125,E2 10007.125} C_VEL
LIN {X 0,Y 402.194,Z 969.694,A -85,B 0,C 180,E1 10016.318,E2 10016.318} C_VEL
LIN {X 0,Y 412.157,Z 925.03,A -85,B 0,C 180,E1 10024.508,E2 10024.508} C_VEL
LIN {X 0,Y 424.831,Z 868.825,A -85,B 0,C 180,E1 10031.025,E2 10031.025} C_VEL
LIN {X 0,Y 436.319,Z 805.459,A -85,B 0,C 180,E1 10035.481,E2 10035.481} C_VEL
LIN {X 0,Y 439.672,Z 771.278,A -85,B 0,C 180,E1 10037.146,E2 10037.146} C_VEL
LIN {X 0,Y 414.213,Z 722.79,A -85,B 0,C 180,E1 10043.339,E2 10043.339} C_VEL
LIN {X 0,Y 393.716,Z 691.44,A -85,B 0,C 180,E1 10049.46,E2 10049.46} C_VEL
LIN {X 0,Y 393.918,Z 691.44,A -85,B 0,C 180,E1 10060.908,E2 10060.908} C_VEL
LIN {X 0,Y 394.784,Z 691.44,A -85,B 0,C 180,E1 10072.286,E2 10072.286} C_VEL
LIN {X 0,Y 395.028,Z 691.44,A -85,B 0,C 180,E1 10081.115,E2 10081.115} C_VEL
LIN {X 0,Y 395.095,Z 693.222,A -85,B 0,C 180,E1 10083.688,E2 10083.688} C_VEL
LIN {X 0,Y 421.285,Z 733.979,A -85,B 0,C 180,E1 10091.043,E2 10091.043} C_VEL
LIN {X 0,Y 438.463,Z 776.381,A -85,B 0,C 180,E1 10096.226,E2 10096.226} C_VEL
LIN {X 0,Y 427.375,Z 837.998,A -85,B 0,C 180,E1 10100.359,E2 10100.359} C_VEL
LIN {X 0,Y 414.792,Z 892.823,A -85,B 0,C 180,E1 10106.483,E2 10106.483} C_VEL
LIN {X 0,Y 404.042,Z 938.159,A -85,B 0,C 180,E1 10114.57,E2 10114.57} C_VEL
LIN {X 0,Y 397.442,Z 970.297,A -85,B 0,C 180,E1 10123.896,E2 10123.896} C_VEL
LIN {X 0,Y 395.249,Z 987.24,A -85,B 0,C 180,E1 10132.672,E2 10132.672} C_VEL
LIN {X 0,Y 394.349,Z 993.141,A -85,B 0,C 180,E1 10141.247,E2 10141.247} C_VEL
LIN {X 0,Y 395.196,Z 988.521,A -85,B 0,C 180,E1 10150.177,E2 10150.177} C_VEL
LIN {X 0,Y 396.81,Z 972.88,A -85,B 0,C 180,E1 10158.976,E2 10158.976} C_VEL
LIN {X 0,Y 402.349,Z 943.444,A -85,B 0,C 180,E1 10168.071,E2 10168.071} C_VEL
LIN {X 0,Y 412.711,Z 900.386,A -85,B 0,C 180,E1 10176.291,E2 10176.291} C_VEL
LIN {X 0,Y 425.655,Z 844.993,A -85,B 0,C 180,E1 10182.876,E2 10182.876} C_VEL
LIN {X 0,Y 436.989,Z 783.507,A -85,B 0,C 180,E1 10187.269,E2 10187.269} C_VEL
LIN {X 0,Y 436.549,Z 769.193,A -85,B 0,C 180,E1 10188.312,E2 10188.312} C_VEL
LIN {X 0,Y 412.452,Z 721.074,A -85,B 0,C 180,E1 10194.537,E2 10194.537} C_VEL
LIN {X 0,Y 393.792,Z 691.44,A -85,B 0,C 180,E1 10199.336,E2 10199.336} C_VEL
LIN {X 0,Y 393.568,Z 691.44,A -85,B 0,C 180,E1 10211.244,E2 10211.244} C_VEL
LIN {X 0,Y 393.482,Z 691.44,A -85,B 0,C 180,E1 10222.247,E2 10222.247} C_VEL
LIN {X 0,Y 393.86,Z 691.44,A -85,B 0,C 180,E1 10233.691,E2 10233.691} C_VEL
LIN {X 0,Y 394.743,Z 691.44,A -85,B 0,C 180,E1 10245.519,E2 10245.519} C_VEL
LIN {X 0,Y 394.916,Z 691.44,A -85,B 0,C 180,E1 10256.682,E2 10256.682} C_VEL
LIN {X 0,Y 394.8,Z 691.44,A -85,B 0,C 180,E1 10265.498,E2 10265.498} C_VEL
LIN {X 0,Y 394.379,Z 691.44,A -85,B 0,C 180,E1 10276.753,E2 10276.753} C_VEL
LIN {X 0,Y 393.944,Z 691.44,A -85,B 0,C 180,E1 10286.269,E2 10286.269} C_VEL
LIN {X 0,Y 393.936,Z 693.473,A -85,B 0,C 180,E1 10292.403,E2 10292.403} C_VEL
LIN {X 0,Y 429.156,Z 749.408,A -85,B 0,C 180,E1 10300.373,E2 10300.373} C_VEL
LIN {X 0,Y 440.388,Z 776.583,A -85,B 0,C 180,E1 10303.205,E2 10303.205} C_VEL
LIN {X 0,Y 430.548,Z 841.673,A -85,B 0,C 180,E1 10306.709,E2 10306.709} C_VEL
LIN {X 0,Y 418.072,Z 900.713,A -85,B 0,C 180,E1 10312.225,E2 10312.225} C_VEL
LIN {X 0,Y 406.314,Z 950.957,A -85,B 0,C 180,E1 10319.719,E2 10319.719} C_VEL
LIN {X 0,Y 398.702,Z 989.098,A -85,B 0,C 180,E1 10328.742,E2 10328.742} C_VEL
LIN {X 0,Y 395.826,Z 1011.888,A -85,B 0,C 180,E1 10337.826,E2 10337.826} C_VEL
LIN {X 0,Y 395.304,Z 1016.34,A -85,B 0,C 180,E1 10340.625,E2 10340.625} C_VEL
LIN {X 0,Y 387.111,Z 1021.047,A -85,B 0,C 180,E1 10345.654,E2 10345.654} C_VEL
LIN {X 0,Y 387.195,Z 1021.654,A -85,B 0,C 180,E1 10353.37,E2 10353.37} C_VEL
LIN {X 0,Y 387.558,Z 1011.51,A -85,B 0,C 180,E1 10362.437,E2 10362.437} C_VEL
LIN {X 0,Y 391.469,Z 986.885,A -85,B 0,C 180,E1 10372.208,E2 10372.208} C_VEL
LIN {X 0,Y 400.108,Z 946.967,A -85,B 0,C 180,E1 10381.477,E2 10381.477} C_VEL
LIN {X 0,Y 412.412,Z 894.911,A -85,B 0,C 180,E1 10389.052,E2 10389.052} C_VEL
LIN {X 0,Y 425.378,Z 835.278,A -85,B 0,C 180,E1 10394.424,E2 10394.424} C_VEL
LIN {X 0,Y 433.791,Z 774.561,A -85,B 0,C 180,E1 10397.788,E2 10397.788} C_VEL
LIN {X 0,Y 409.717,Z 727.679,A -85,B 0,C 180,E1 10404.057,E2 10404.057} C_VEL
LIN {X 0,Y 388.43,Z 697.465,A -85,B 0,C 180,E1 10410.523,E2 10410.523} C_VEL
LIN {X 0,Y 385.71,Z 691.44,A -85,B 0,C 180,E1 10412.284,E2 10412.284} C_VEL
LIN {X 0,Y 386.085,Z 691.44,A -85,B 0,C 180,E1 10424.369,E2 10424.369} C_VEL
LIN {X 0,Y 386.78,Z 691.44,A -85,B 0,C 180,E1 10434.388,E2 10434.388} C_VEL
LIN {X 0,Y 387.205,Z 693.168,A -85,B 0,C 180,E1 10441.332,E2 10441.332} C_VEL
LIN {X 0,Y 409.251,Z 726.128,A -85,B 0,C 180,E1 10448.388,E2 10448.388} C_VEL
LIN {X 0,Y 430.555,Z 771.574,A -85,B 0,C 180,E1 10454.775,E2 10454.775} C_VEL
LIN {X 0,Y 431.843,Z 783.304,A -85,B 0,C 180,E1 10455.813,E2 10455.813} C_VEL
LIN {X 0,Y 419.924,Z 844.598,A -85,B 0,C 180,E1 10460.181,E2 10460.181} C_VEL
LIN {X 0,Y 406.368,Z 899.721,A -85,B 0,C 180,E1 10466.78,E2 10466.78} C_VEL
LIN {X 0,Y 395.325,Z 943.628,A -85,B 0,C 180,E1 10475.263,E2 10475.263} C_VEL
LIN {X 0,Y 389.089,Z 973.124,A -85,B 0,C 180,E1 10484.521,E2 10484.521} C_VEL
LIN {X 0,Y 387.144,Z 988.751,A -85,B 0,C 180,E1 10493.473,E2 10493.473} C_VEL
LIN {X 0,Y 386.358,Z 993.377,A -85,B 0,C 180,E1 10503.147,E2 10503.147} C_VEL
LIN {X 0,Y 387.27,Z 987.119,A -85,B 0,C 180,E1 10511.731,E2 10511.731} C_VEL
LIN {X 0,Y 389.677,Z 968.812,A -85,B 0,C 180,E1 10521.038,E2 10521.038} C_VEL
LIN {X 0,Y 396.715,Z 936.567,A -85,B 0,C 180,E1 10530.274,E2 10530.274} C_VEL
LIN {X 0,Y 408.731,Z 889.607,A -85,B 0,C 180,E1 10538.541,E2 10538.541} C_VEL
LIN {X 0,Y 422.182,Z 832.666,A -85,B 0,C 180,E1 10544.707,E2 10544.707} C_VEL
LIN {X 0,Y 431.211,Z 774.315,A -85,B 0,C 180,E1 10548.712,E2 10548.712} C_VEL
LIN {X 0,Y 408.1,Z 726.746,A -85,B 0,C 180,E1 10555.051,E2 10555.051} C_VEL
LIN {X 0,Y 385.743,Z 691.44,A -85,B 0,C 180,E1 10561.09,E2 10561.09} C_VEL
LIN {X 0,Y 385.526,Z 691.44,A -85,B 0,C 180,E1 10570.505,E2 10570.505} C_VEL
LIN {X 0,Y 385.508,Z 691.44,A -85,B 0,C 180,E1 10580.143,E2 10580.143} C_VEL
LIN {X 0,Y 385.722,Z 691.44,A -85,B 0,C 180,E1 10590.535,E2 10590.535} C_VEL
LIN {X 0,Y 386.332,Z 691.44,A -85,B 0,C 180,E1 10602.856,E2 10602.856} C_VEL
LIN {X 0,Y 386.811,Z 691.44,A -85,B 0,C 180,E1 10612.095,E2 10612.095} C_VEL
LIN {X 0,Y 387.035,Z 691.44,A -85,B 0,C 180,E1 10623.355,E2 10623.355} C_VEL
LIN {X 0,Y 386.451,Z 691.44,A -85,B 0,C 180,E1 10634.767,E2 10634.767} C_VEL
LIN {X 0,Y 385.995,Z 691.44,A -85,B 0,C 180,E1 10644.356,E2 10644.356} C_VEL
LIN {X 0,Y 385.801,Z 692.778,A -85,B 0,C 180,E1 10650.627,E2 10650.627} C_VEL
LIN {X 0,Y 421.678,Z 749.606,A -85,B 0,C 180,E1 10659.248,E2 10659.248} C_VEL
LIN {X 0,Y 434.37,Z 779.457,A -85,B 0,C 180,E1 10662.56,E2 10662.56} C_VEL
LIN {X 0,Y 424.109,Z 843.333,A -85,B 0,C 180,E1 10666.108,E2 10666.108} C_VEL
LIN {X 0,Y 410.918,Z 902.912,A -85,B 0,C 180,E1 10671.821,E2 10671.821} C_VEL
LIN {X 0,Y 398.387,Z 953.594,A -85,B 0,C 180,E1 10679.686,E2 10679.686} C_VEL
LIN {X 0,Y 390.922,Z 988.959,A -85,B 0,C 180,E1 10688.358,E2 10688.358} C_VEL
LIN {X 0,Y 387.801,Z 1012.607,A -85,B 0,C 180,E1 10698.161,E2 10698.161} C_VEL
LIN {X 0,Y 387.111,Z 1021.047,A -85,B 0,C 180,E1 10705.654,E2 10705.654} C_VEL
LIN {X 0,Y 379.262,Z 1022.073,A -85,B 0,C 180,E1 10710.838,E2 10710.838} C_VEL
LIN {X 0,Y 379.306,Z 1014.841,A -85,B 0,C 180,E1 10720.372,E2 10720.372} C_VEL
LIN {X 0,Y 381.771,Z 995.389,A -85,B 0,C 180,E1 10729.748,E2 10729.748} C_VEL
LIN {X 0,Y 388.56,Z 963.187,A -85,B 0,C 180,E1 10738.756,E2 10738.756} C_VEL
LIN {X 0,Y 400.785,Z 915.061,A -85,B 0,C 180,E1 10747.197,E2 10747.197} C_VEL
LIN {X 0,Y 414.899,Z 857.273,A -85,B 0,C 180,E1 10753.48,E2 10753.48} C_VEL
LIN {X 0,Y 426.776,Z 795.243,A -85,B 0,C 180,E1 10757.506,E2 10757.506} C_VEL
LIN {X 0,Y 427.743,Z 777.431,A -85,B 0,C 180,E1 10758.506,E2 10758.506} C_VEL
LIN {X 0,Y 404.408,Z 730.759,A -85,B 0,C 180,E1 10765.054,E2 10765.054} C_VEL
LIN {X 0,Y 382.043,Z 698.55,A -85,B 0,C 180,E1 10772.634,E2 10772.634} C_VEL
LIN {X 0,Y 377.693,Z 691.44,A -85,B 0,C 180,E1 10775.073,E2 10775.073} C_VEL
LIN {X 0,Y 378.148,Z 691.44,A -85,B 0,C 180,E1 10784.901,E2 10784.901} C_VEL
LIN {X 0,Y 379.008,Z 691.44,A -85,B 0,C 180,E1 10796.574,E2 10796.574} C_VEL
LIN {X 0,Y 379.791,Z 693.841,A -85,B 0,C 180,E1 10798.685,E2 10798.685} C_VEL
LIN {X 0,Y 399.463,Z 722.087,A -85,B 0,C 180,E1 10806.01,E2 10806.01} C_VEL
LIN {X 0,Y 420.18,Z 762.829,A -85,B 0,C 180,E1 10812.526,E2 10812.526} C_VEL
LIN {X 0,Y 426.114,Z 784.996,A -85,B 0,C 180,E1 10815.105,E2 10815.105} C_VEL
LIN {X 0,Y 413.65,Z 845.873,A -85,B 0,C 180,E1 10819.522,E2 10819.522} C_VEL
LIN {X 0,Y 399.44,Z 900.846,A -85,B 0,C 180,E1 10826.225,E2 10826.225} C_VEL
LIN {X 0,Y 388.211,Z 943.169,A -85,B 0,C 180,E1 10834.534,E2 10834.534} C_VEL
LIN {X 0,Y 381.339,Z 973.399,A -85,B 0,C 180,E1 10844.144,E2 10844.144} C_VEL
LIN {X 0,Y 379.159,Z 989.303,A -85,B 0,C 180,E1 10853.555,E2 10853.555} C_VEL
LIN {X 0,Y 378.328,Z 993.763,A -85,B 0,C 180,E1 10862.529,E2 10862.529} C_VEL
LIN {X 0,Y 379.276,Z 988.171,A -85,B 0,C 180,E1 10871.339,E2 10871.339} C_VEL
LIN {X 0,Y 381.359,Z 972.102,A -85,B 0,C 180,E1 10880.263,E2 10880.263} C_VEL
LIN {X 0,Y 388.082,Z 941.624,A -85,B 0,C 180,E1 10889.72,E2 10889.72} C_VEL
LIN {X 0,Y 399.614,Z 898.869,A -85,B 0,C 180,E1 10897.913,E2 10897.913} C_VEL
LIN {X 0,Y 413.723,Z 843.984,A -85,B 0,C 180,E1 10904.472,E2 10904.472} C_VEL
LIN {X 0,Y 426.004,Z 781.858,A -85,B 0,C 180,E1 10908.888,E2 10908.888} C_VEL
LIN {X 0,Y 407.543,Z 738.92,A -85,B 0,C 180,E1 10914.558,E2 10914.558} C_VEL
LIN {X 0,Y 379.432,Z 696.463,A -85,B 0,C 180,E1 10922.068,E2 10922.068} C_VEL
LIN {X 0,Y 377.565,Z 691.44,A -85,B 0,C 180,E1 10922.863,E2 10922.863} C_VEL
LIN {X 0,Y 377.415,Z 691.44,A -85,B 0,C 180,E1 10934.723,E2 10934.723} C_VEL
LIN {X 0,Y 377.494,Z 691.44,A -85,B 0,C 180,E1 10945.502,E2 10945.502} C_VEL
LIN {X 0,Y 377.705,Z 691.44,A -85,B 0,C 180,E1 10955.039,E2 10955.039} C_VEL
LIN {X 0,Y 378.689,Z 691.44,A -85,B 0,C 180,E1 10967.255,E2 10967.255} C_VEL
LIN {X 0,Y 379.034,Z 691.44,A -85,B 0,C 180,E1 10978.991,E2 10978.991} C_VEL
LIN {X 0,Y 378.672,Z 691.44,A -85,B 0,C 180,E1 10990.37,E2 10990.37} C_VEL
LIN {X 0,Y 378.069,Z 691.44,A -85,B 0,C 180,E1 11002.391,E2 11002.391} C_VEL
LIN {X 0,Y 378.023,Z 693.481,A -85,B 0,C 180,E1 11008.842,E2 11008.842} C_VEL
LIN {X 0,Y 412.655,Z 746.924,A -85,B 0,C 180,E1 11017.683,E2 11017.683} C_VEL
LIN {X 0,Y 428.397,Z 782.374,A -85,B 0,C 180,E1 11021.899,E2 11021.899} C_VEL
LIN {X 0,Y 417.117,Z 847.985,A -85,B 0,C 180,E1 11025.725,E2 11025.725} C_VEL
LIN {X 0,Y 403.761,Z 904.872,A -85,B 0,C 180,E1 11031.388,E2 11031.388} C_VEL
LIN {X 0,Y 390.823,Z 954.729,A -85,B 0,C 180,E1 11039.359,E2 11039.359} C_VEL
LIN {X 0,Y 382.837,Z 990.704,A -85,B 0,C 180,E1 11048.584,E2 11048.584} C_VEL
LIN {X 0,Y 379.727,Z 1013.811,A -85,B 0,C 180,E1 11058.838,E2 11058.838} C_VEL
LIN {X 0,Y 379.127,Z 1021.363,A -85,B 0,C 180,E1 11066.557,E2 11066.557} C_VEL
LIN {X 0,Y 379.262,Z 1022.073,A -85,B 0,C 180,E1 11070.838,E2 11070.838} C_VEL
LIN {X 0,Y 371.218,Z 1019.416,A -85,B 0,C 180,E1 11076.108,E2 11076.108} C_VEL
LIN {X 0,Y 372.863,Z 1004.615,A -85,B 0,C 180,E1 11086.255,E2 11086.255} C_VEL
LIN {X 0,Y 378.538,Z 974.203,A -85,B 0,C 180,E1 11096.572,E2 11096.572} C_VEL
LIN {X 0,Y 389.881,Z 930.326,A -85,B 0,C 180,E1 11105.559,E2 11105.559} C_VEL
LIN {X 0,Y 404.371,Z 875.818,A -85,B 0,C 180,E1 11112.536,E2 11112.536} C_VEL
LIN {X 0,Y 418.263,Z 811.774,A -85,B 0,C 180,E1 11117.476,E2 11117.476} C_VEL
LIN {X 0,Y 422.181,Z 781.37,A -85,B 0,C 180,E1 11119.124,E2 11119.124} C_VEL
LIN {X 0,Y 400.277,Z 736.144,A -85,B 0,C 180,E1 11125.751,E2 11125.751} C_VEL
LIN {X 0,Y 379.629,Z 705.807,A -85,B 0,C 180,E1 11133.141,E2 11133.141} C_VEL
LIN {X 0,Y 371.43,Z 696.374,A -85,B 0,C 180,E1 11137.668,E2 11137.668} C_VEL
LIN {X 0,Y 369.744,Z 691.44,A -85,B 0,C 180,E1 11139.606,E2 11139.606} C_VEL
LIN {X 0,Y 370.676,Z 691.44,A -85,B 0,C 180,E1 11151.781,E2 11151.781} C_VEL
LIN {X 0,Y 371.116,Z 693.731,A -85,B 0,C 180,E1 11154.349,E2 11154.349} C_VEL
LIN {X 0,Y 378.96,Z 703.562,A -85,B 0,C 180,E1 11158.914,E2 11158.914} C_VEL
LIN {X 0,Y 397.763,Z 731.157,A -85,B 0,C 180,E1 11166.104,E2 11166.104} C_VEL
LIN {X 0,Y 417.503,Z 774.198,A -85,B 0,C 180,E1 11172.903,E2 11172.903} C_VEL
LIN {X 0,Y 420.093,Z 788.921,A -85,B 0,C 180,E1 11174.5,E2 11174.5} C_VEL
LIN {X 0,Y 407.137,Z 848.31,A -85,B 0,C 180,E1 11178.956,E2 11178.956} C_VEL
LIN {X 0,Y 392.478,Z 902.287,A -85,B 0,C 180,E1 11185.698,E2 11185.698} C_VEL
LIN {X 0,Y 380.26,Z 945.689,A -85,B 0,C 180,E1 11194.518,E2 11194.518} C_VEL
LIN {X 0,Y 373.104,Z 975.587,A -85,B 0,C 180,E1 11204.618,E2 11204.618} C_VEL
LIN {X 0,Y 371.151,Z 989.857,A -85,B 0,C 180,E1 11213.638,E2 11213.638} C_VEL
LIN {X 0,Y 370.296,Z 994.131,A -85,B 0,C 180,E1 11221.881,E2 11221.881} C_VEL
LIN {X 0,Y 371.264,Z 989.077,A -85,B 0,C 180,E1 11230.986,E2 11230.986} C_VEL
LIN {X 0,Y 373.57,Z 972.4,A -85,B 0,C 180,E1 11240.649,E2 11240.649} C_VEL
LIN {X 0,Y 380.89,Z 941.603,A -85,B 0,C 180,E1 11250.36,E2 11250.36} C_VEL
LIN {X 0,Y 392.946,Z 899.094,A -85,B 0,C 180,E1 11258.607,E2 11258.607} C_VEL
LIN {X 0,Y 407.677,Z 844.11,A -85,B 0,C 180,E1 11265.243,E2 11265.243} C_VEL
LIN {X 0,Y 419.158,Z 780.94,A -85,B 0,C 180,E1 11269.953,E2 11269.953} C_VEL
LIN {X 0,Y 396.921,Z 733.682,A -85,B 0,C 180,E1 11276.793,E2 11276.793} C_VEL
LIN {X 0,Y 369.5,Z 691.44,A -85,B 0,C 180,E1 11285.027,E2 11285.027} C_VEL
LIN {X 0,Y 369.335,Z 691.44,A -85,B 0,C 180,E1 11295.979,E2 11295.979} C_VEL
LIN {X 0,Y 369.522,Z 691.44,A -85,B 0,C 180,E1 11307.344,E2 11307.344} C_VEL
LIN {X 0,Y 369.77,Z 691.44,A -85,B 0,C 180,E1 11317.434,E2 11317.434} C_VEL
LIN {X 0,Y 370.643,Z 691.44,A -85,B 0,C 180,E1 11326.974,E2 11326.974} C_VEL
LIN {X 0,Y 371.055,Z 691.44,A -85,B 0,C 180,E1 11339.003,E2 11339.003} C_VEL
LIN {X 0,Y 370.65,Z 691.44,A -85,B 0,C 180,E1 11350.597,E2 11350.597} C_VEL
LIN {X 0,Y 370.024,Z 691.44,A -85,B 0,C 180,E1 11362.66,E2 11362.66} C_VEL
LIN {X 0,Y 369.936,Z 693.107,A -85,B 0,C 180,E1 11366.796,E2 11366.796} C_VEL
LIN {X 0,Y 404.209,Z 745.266,A -85,B 0,C 180,E1 11376.152,E2 11376.152} C_VEL
LIN {X 0,Y 422.606,Z 784.416,A -85,B 0,C 180,E1 11381.192,E2 11381.192} C_VEL
LIN {X 0,Y 410.451,Z 850.859,A -85,B 0,C 180,E1 11385.185,E2 11385.185} C_VEL
LIN {X 0,Y 396.456,Z 907.453,A -85,B 0,C 180,E1 11391.036,E2 11391.036} C_VEL
LIN {X 0,Y 383.146,Z 956.198,A -85,B 0,C 180,E1 11399.097,E2 11399.097} C_VEL
LIN {X 0,Y 374.808,Z 992.025,A -85,B 0,C 180,E1 11408.675,E2 11408.675} C_VEL
LIN {X 0,Y 371.752,Z 1013.656,A -85,B 0,C 180,E1 11418.704,E2 11418.704} C_VEL
LIN {X 0,Y 371.125,Z 1021.065,A -85,B 0,C 180,E1 11426.483,E2 11426.483} C_VEL
LIN {X 0,Y 371.18,Z 1021.043,A -85,B 0,C 180,E1 11433.516,E2 11433.516} C_VEL
LIN {X 0,Y 371.218,Z 1019.416,A -85,B 0,C 180,E1 11436.108,E2 11436.108} C_VEL
LIN {X 0,Y 363.384,Z 1013.361,A -85,B 0,C 180,E1 11441.453,E2 11441.453} C_VEL
LIN {X 0,Y 366.58,Z 993.443,A -85,B 0,C 180,E1 11451.1,E2 11451.1} C_VEL
LIN {X 0,Y 375.651,Z 956.706,A -85,B 0,C 180,E1 11461.249,E2 11461.249} C_VEL
LIN {X 0,Y 389.203,Z 908.64,A -85,B 0,C 180,E1 11469.459,E2 11469.459} C_VEL
LIN {X 0,Y 404.566,Z 850.705,A -85,B 0,C 180,E1 11475.588,E2 11475.588} C_VEL
LIN {X 0,Y 416.305,Z 784.445,A -85,B 0,C 180,E1 11479.85,E2 11479.85} C_VEL
LIN {X 0,Y 395.999,Z 741.349,A -85,B 0,C 180,E1 11486.466,E2 11486.466} C_VEL
LIN {X 0,Y 377.101,Z 712.806,A -85,B 0,C 180,E1 11493.753,E2 11493.753} C_VEL
LIN {X 0,Y 366.992,Z 698.954,A -85,B 0,C 180,E1 11500.713,E2 11500.713} C_VEL
LIN {X 0,Y 366.999,Z 698.554,A -85,B 0,C 180,E1 11511.698,E2 11511.698} C_VEL
LIN {X 0,Y 375.845,Z 708.772,A -85,B 0,C 180,E1 11517.919,E2 11517.919} C_VEL
LIN {X 0,Y 394.8,Z 738.727,A -85,B 0,C 180,E1 11525.83,E2 11525.83} C_VEL
LIN {X 0,Y 413.133,Z 781.47,A -85,B 0,C 180,E1 11532.742,E2 11532.742} C_VEL
LIN {X 0,Y 413.94,Z 793.661,A -85,B 0,C 180,E1 11533.926,E2 11533.926} C_VEL
LIN {X 0,Y 399.836,Z 854.105,A -85,B 0,C 180,E1 11538.712,E2 11538.712} C_VEL
LIN {X 0,Y 384.457,Z 906.952,A -85,B 0,C 180,E1 11545.7,E2 11545.7} C_VEL
LIN {X 0,Y 372.086,Z 948.88,A -85,B 0,C 180,E1 11554.703,E2 11554.703} C_VEL
LIN {X 0,Y 364.997,Z 977.395,A -85,B 0,C 180,E1 11564.938,E2 11564.938} C_VEL
LIN {X 0,Y 363.016,Z 991.286,A -85,B 0,C 180,E1 11574.606,E2 11574.606} C_VEL
LIN {X 0,Y 362.393,Z 994.116,A -85,B 0,C 180,E1 11584.2,E2 11584.2} C_VEL
LIN {X 0,Y 363.573,Z 986.826,A -85,B 0,C 180,E1 11593.264,E2 11593.264} C_VEL
LIN {X 0,Y 367.693,Z 965.933,A -85,B 0,C 180,E1 11603.683,E2 11603.683} C_VEL
LIN {X 0,Y 377.192,Z 931.037,A -85,B 0,C 180,E1 11613.46,E2 11613.46} C_VEL
LIN {X 0,Y 390.794,Z 884.364,A -85,B 0,C 180,E1 11621.48,E2 11621.48} C_VEL
LIN {X 0,Y 405.819,Z 827.118,A -85,B 0,C 180,E1 11627.52,E2 11627.52} C_VEL
LIN {X 0,Y 413.255,Z 784.558,A -85,B 0,C 180,E1 11630.553,E2 11630.553} C_VEL
LIN {X 0,Y 391.439,Z 737.228,A -85,B 0,C 180,E1 11637.668,E2 11637.668} C_VEL
LIN {X 0,Y 363.787,Z 697.12,A -85,B 0,C 180,E1 11646.055,E2 11646.055} C_VEL
LIN {X 0,Y 361.287,Z 691.44,A -85,B 0,C 180,E1 11647.523,E2 11647.523} C_VEL
LIN {X 0,Y 361.326,Z 691.44,A -85,B 0,C 180,E1 11659.378,E2 11659.378} C_VEL
LIN {X 0,Y 361.561,Z 691.44,A -85,B 0,C 180,E1 11671.131,E2 11671.131} C_VEL
LIN {X 0,Y 362.032,Z 691.44,A -85,B 0,C 180,E1 11681.666,E2 11681.666} C_VEL
LIN {X 0,Y 362.751,Z 691.44,A -85,B 0,C 180,E1 11691.567,E2 11691.567} C_VEL
LIN {X 0,Y 363.447,Z 691.44,A -85,B 0,C 180,E1 11701.18,E2 11701.18} C_VEL
LIN {X 0,Y 362.427,Z 691.44,A -85,B 0,C 180,E1 11713.293,E2 11713.293} C_VEL
LIN {X 0,Y 361.963,Z 692.925,A -85,B 0,C 180,E1 11724.596,E2 11724.596} C_VEL
LIN {X 0,Y 395.102,Z 742.58,A -85,B 0,C 180,E1 11734.343,E2 11734.343} C_VEL
LIN {X 0,Y 416.646,Z 787.209,A -85,B 0,C 180,E1 11740.508,E2 11740.508} C_VEL
LIN {X 0,Y 404.073,Z 852.853,A -85,B 0,C 180,E1 11744.566,E2 11744.566} C_VEL
LIN {X 0,Y 388.861,Z 911.004,A -85,B 0,C 180,E1 11750.799,E2 11750.799} C_VEL
LIN {X 0,Y 375.219,Z 958.577,A -85,B 0,C 180,E1 11759.053,E2 11759.053} C_VEL
LIN {X 0,Y 366.742,Z 993.712,A -85,B 0,C 180,E1 11768.907,E2 11768.907} C_VEL
LIN {X 0,Y 363.63,Z 1014.315,A -85,B 0,C 180,E1 11779.175,E2 11779.175} C_VEL
LIN {X 0,Y 363,Z 1021.469,A -85,B 0,C 180,E1 11788.802,E2 11788.802} C_VEL
LIN {X 0,Y 363.385,Z 1017.126,A -85,B 0,C 180,E1 11798.404,E2 11798.404} C_VEL
LIN {X 0,Y 363.384,Z 1013.361,A -85,B 0,C 180,E1 11801.453,E2 11801.453} C_VEL
LIN {X 0,Y 356.996,Z 1004.224,A -85,B 0,C 180,E1 11806.841,E2 11806.841} C_VEL
LIN {X 0,Y 363.203,Z 974.89,A -85,B 0,C 180,E1 11817.362,E2 11817.362} C_VEL
LIN {X 0,Y 375.558,Z 932.331,A -85,B 0,C 180,E1 11826.586,E2 11826.586} C_VEL
LIN {X 0,Y 391.598,Z 878.057,A -85,B 0,C 180,E1 11833.875,E2 11833.875} C_VEL
LIN {X 0,Y 406.767,Z 814.642,A -85,B 0,C 180,E1 11838.966,E2 11838.966} C_VEL
LIN {X 0,Y 410.845,Z 788.576,A -85,B 0,C 180,E1 11840.453,E2 11840.453} C_VEL
LIN {X 0,Y 391.825,Z 746.418,A -85,B 0,C 180,E1 11847.195,E2 11847.195} C_VEL
LIN {X 0,Y 374.603,Z 719.664,A -85,B 0,C 180,E1 11854.371,E2 11854.371} C_VEL
LIN {X 0,Y 365.212,Z 706.557,A -85,B 0,C 180,E1 11861.452,E2 11861.452} C_VEL
LIN {X 0,Y 366.749,Z 706.846,A -85,B 0,C 180,E1 11872.497,E2 11872.497} C_VEL
LIN {X 0,Y 377.404,Z 721.426,A -85,B 0,C 180,E1 11879.415,E2 11879.415} C_VEL
LIN {X 0,Y 395.976,Z 754.914,A -85,B 0,C 180,E1 11887.257,E2 11887.257} C_VEL
LIN {X 0,Y 408.977,Z 792.65,A -85,B 0,C 180,E1 11892.998,E2 11892.998} C_VEL
LIN {X 0,Y 394.579,Z 852.104,A -85,B 0,C 180,E1 11897.653,E2 11897.653} C_VEL
LIN {X 0,Y 378.442,Z 905.652,A -85,B 0,C 180,E1 11904.686,E2 11904.686} C_VEL
LIN {X 0,Y 365.075,Z 948.439,A -85,B 0,C 180,E1 11913.896,E2 11913.896} C_VEL
LIN {X 0,Y 357.231,Z 977.602,A -85,B 0,C 180,E1 11924.507,E2 11924.507} C_VEL
LIN {X 0,Y 355.131,Z 990.884,A -85,B 0,C 180,E1 11933.697,E2 11933.697} C_VEL
LIN {X 0,Y 354.264,Z 994.555,A -85,B 0,C 180,E1 11943.27,E2 11943.27} C_VEL
LIN {X 0,Y 355.477,Z 988.261,A -85,B 0,C 180,E1 11952.593,E2 11952.593} C_VEL
LIN {X 0,Y 359.229,Z 969.057,A -85,B 0,C 180,E1 11963.076,E2 11963.076} C_VEL
LIN {X 0,Y 368.85,Z 935.093,A -85,B 0,C 180,E1 11973.244,E2 11973.244} C_VEL
LIN {X 0,Y 382.661,Z 890.433,A -85,B 0,C 180,E1 11981.438,E2 11981.438} C_VEL
LIN {X 0,Y 398.789,Z 832.627,A -85,B 0,C 180,E1 11987.898,E2 11987.898} C_VEL
LIN {X 0,Y 407.262,Z 787.791,A -85,B 0,C 180,E1 11991.223,E2 11991.223} C_VEL
LIN {X 0,Y 386.206,Z 741.425,A -85,B 0,C 180,E1 11998.474,E2 11998.474} C_VEL
LIN {X 0,Y 360.325,Z 703.147,A -85,B 0,C 180,E1 12006.782,E2 12006.782} C_VEL
LIN {X 0,Y 353.283,Z 691.44,A -85,B 0,C 180,E1 12009.653,E2 12009.653} C_VEL
LIN {X 0,Y 353.237,Z 691.44,A -85,B 0,C 180,E1 12021.463,E2 12021.463} C_VEL
LIN {X 0,Y 353.531,Z 691.44,A -85,B 0,C 180,E1 12033.201,E2 12033.201} C_VEL
LIN {X 0,Y 354.434,Z 691.44,A -85,B 0,C 180,E1 12044.45,E2 12044.45} C_VEL
LIN {X 0,Y 354.927,Z 691.44,A -85,B 0,C 180,E1 12056.307,E2 12056.307} C_VEL
LIN {X 0,Y 354.729,Z 691.44,A -85,B 0,C 180,E1 12066.121,E2 12066.121} C_VEL
LIN {X 0,Y 354.248,Z 691.44,A -85,B 0,C 180,E1 12076.145,E2 12076.145} C_VEL
LIN {X 0,Y 354.093,Z 693.335,A -85,B 0,C 180,E1 12082.229,E2 12082.229} C_VEL
LIN {X 0,Y 384.465,Z 737.399,A -85,B 0,C 180,E1 12091.937,E2 12091.937} C_VEL
LIN {X 0,Y 409.534,Z 786.521,A -85,B 0,C 180,E1 12099.367,E2 12099.367} C_VEL
LIN {X 0,Y 408.653,Z 802.588,A -85,B 0,C 180,E1 12100.421,E2 12100.421} C_VEL
LIN {X 0,Y 394.39,Z 867.022,A -85,B 0,C 180,E1 12104.994,E2 12104.994} C_VEL
LIN {X 0,Y 378.546,Z 923.742,A -85,B 0,C 180,E1 12111.947,E2 12111.947} C_VEL
LIN {X 0,Y 365.458,Z 968.314,A -85,B 0,C 180,E1 12120.81,E2 12120.81} C_VEL
LIN {X 0,Y 358.006,Z 999.34,A -85,B 0,C 180,E1 12130.82,E2 12130.82} C_VEL
LIN {X 0,Y 355.22,Z 1016.894,A -85,B 0,C 180,E1 12141.4,E2 12141.4} C_VEL
LIN {X 0,Y 355.361,Z 1021.172,A -85,B 0,C 180,E1 12151.223,E2 12151.223} C_VEL
LIN {X 0,Y 355.366,Z 1013.882,A -85,B 0,C 180,E1 12161.079,E2 12161.079} C_VEL
LIN {X 0,Y 356.996,Z 1004.224,A -85,B 0,C 180,E1 12166.841,E2 12166.841} C_VEL
LIN {X 0,Y 351.327,Z 992.454,A -85,B 0,C 180,E1 12172.181,E2 12172.181} C_VEL
LIN {X 0,Y 361.409,Z 956.295,A -85,B 0,C 180,E1 12182.55,E2 12182.55} C_VEL
LIN {X 0,Y 376.553,Z 907.745,A -85,B 0,C 180,E1 12191.103,E2 12191.103} C_VEL
LIN {X 0,Y 393.283,Z 850.053,A -85,B 0,C 180,E1 12197.314,E2 12197.314} C_VEL
LIN {X 0,Y 405.429,Z 792.729,A -85,B 0,C 180,E1 12201.076,E2 12201.076} C_VEL
LIN {X 0,Y 387.678,Z 751.411,A -85,B 0,C 180,E1 12207.953,E2 12207.953} C_VEL
LIN {X 0,Y 371.7,Z 725.997,A -85,B 0,C 180,E1 12215.207,E2 12215.207} C_VEL
LIN {X 0,Y 363.831,Z 714.33,A -85,B 0,C 180,E1 12221.794,E2 12221.794} C_VEL
LIN {X 0,Y 365.935,Z 715.023,A -85,B 0,C 180,E1 12232.819,E2 12232.819} C_VEL
LIN {X 0,Y 376.169,Z 731.279,A -85,B 0,C 180,E1 12239.703,E2 12239.703} C_VEL
LIN {X 0,Y 392.126,Z 761.61,A -85,B 0,C 180,E1 12246.902,E2 12246.902} C_VEL
LIN {X 0,Y 402.968,Z 796.793,A -85,B 0,C 180,E1 12252.354,E2 12252.354} C_VEL
LIN {X 0,Y 387.594,Z 856.988,A -85,B 0,C 180,E1 12257.276,E2 12257.276} C_VEL
LIN {X 0,Y 370.707,Z 909.456,A -85,B 0,C 180,E1 12264.511,E2 12264.511} C_VEL
LIN {X 0,Y 357.536,Z 949.555,A -85,B 0,C 180,E1 12273.504,E2 12273.504} C_VEL
LIN {X 0,Y 349.404,Z 978.153,A -85,B 0,C 180,E1 12284.222,E2 12284.222} C_VEL
LIN {X 0,Y 347.111,Z 991.633,A -85,B 0,C 180,E1 12293.983,E2 12293.983} C_VEL
LIN {X 0,Y 346.285,Z 994.764,A -85,B 0,C 180,E1 12303.947,E2 12303.947} C_VEL
LIN {X 0,Y 347.669,Z 987.722,A -85,B 0,C 180,E1 12313.518,E2 12313.518} C_VEL
LIN {X 0,Y 352.291,Z 967.076,A -85,B 0,C 180,E1 12324.438,E2 12324.438} C_VEL
LIN {X 0,Y 363.135,Z 931.556,A -85,B 0,C 180,E1 12334.795,E2 12334.795} C_VEL
LIN {X 0,Y 378.122,Z 884.727,A -85,B 0,C 180,E1 12343.048,E2 12343.048} C_VEL
LIN {X 0,Y 394.171,Z 828.34,A -85,B 0,C 180,E1 12349.103,E2 12349.103} C_VEL
LIN {X 0,Y 401.385,Z 791.299,A -85,B 0,C 180,E1 12351.874,E2 12351.874} C_VEL
LIN {X 0,Y 380.773,Z 745.255,A -85,B 0,C 180,E1 12359.385,E2 12359.385} C_VEL
LIN {X 0,Y 354.741,Z 705.586,A -85,B 0,C 180,E1 12368.34,E2 12368.34} C_VEL
LIN {X 0,Y 345.232,Z 691.44,A -85,B 0,C 180,E1 12372.358,E2 12372.358} C_VEL
LIN {X 0,Y 345.306,Z 691.44,A -85,B 0,C 180,E1 12384.397,E2 12384.397} C_VEL
LIN {X 0,Y 345.536,Z 691.44,A -85,B 0,C 180,E1 12395.33,E2 12395.33} C_VEL
LIN {X 0,Y 346.493,Z 691.44,A -85,B 0,C 180,E1 12406.048,E2 12406.048} C_VEL
LIN {X 0,Y 346.912,Z 691.44,A -85,B 0,C 180,E1 12416.222,E2 12416.222} C_VEL
LIN {X 0,Y 346.709,Z 691.44,A -85,B 0,C 180,E1 12426.263,E2 12426.263} C_VEL
LIN {X 0,Y 346.178,Z 691.44,A -85,B 0,C 180,E1 12436.532,E2 12436.532} C_VEL
LIN {X 0,Y 346.26,Z 693.578,A -85,B 0,C 180,E1 12439.598,E2 12439.598} C_VEL
LIN {X 0,Y 373.921,Z 732.689,A -85,B 0,C 180,E1 12449.366,E2 12449.366} C_VEL
LIN {X 0,Y 399.795,Z 780.646,A -85,B 0,C 180,E1 12457.364,E2 12457.364} C_VEL
LIN {X 0,Y 404.289,Z 796.624,A -85,B 0,C 180,E1 12459.267,E2 12459.267} C_VEL
LIN {X 0,Y 389.681,Z 862.28,A -85,B 0,C 180,E1 12463.759,E2 12463.759} C_VEL
LIN {X 0,Y 373.776,Z 917.332,A -85,B 0,C 180,E1 12470.237,E2 12470.237} C_VEL
LIN {X 0,Y 359.279,Z 963.714,A -85,B 0,C 180,E1 12479.06,E2 12479.06} C_VEL
LIN {X 0,Y 350.506,Z 997.477,A -85,B 0,C 180,E1 12489.734,E2 12489.734} C_VEL
LIN {X 0,Y 347.441,Z 1015.488,A -85,B 0,C 180,E1 12500.083,E2 12500.083} C_VEL
LIN {X 0,Y 347.013,Z 1020.873,A -85,B 0,C 180,E1 12508.747,E2 12508.747} C_VEL
LIN {X 0,Y 347.363,Z 1016.497,A -85,B 0,C 180,E1 12518.795,E2 12518.795} C_VEL
LIN {X 0,Y 349.501,Z 1000.13,A -85,B 0,C 180,E1 12529.005,E2 12529.005} C_VEL
LIN {X 0,Y 351.327,Z 992.454,A -85,B 0,C 180,E1 12532.181,E2 12532.181} C_VEL
LIN {X 0,Y 347.36,Z 978.094,A -85,B 0,C 180,E1 12537.49,E2 12537.49} C_VEL
LIN {X 0,Y 361.087,Z 935.164,A -85,B 0,C 180,E1 12547.546,E2 12547.546} C_VEL
LIN {X 0,Y 378.811,Z 880.856,A -85,B 0,C 180,E1 12555.235,E2 12555.235} C_VEL
LIN {X 0,Y 395.385,Z 818.623,A -85,B 0,C 180,E1 12560.487,E2 12560.487} C_VEL
LIN {X 0,Y 399.481,Z 795.021,A -85,B 0,C 180,E1 12561.977,E2 12561.977} C_VEL
LIN {X 0,Y 382.681,Z 755.29,A -85,B 0,C 180,E1 12569.022,E2 12569.022} C_VEL
LIN {X 0,Y 367.727,Z 729.484,A -85,B 0,C 180,E1 12576.944,E2 12576.944} C_VEL
LIN {X 0,Y 361.863,Z 721.752,A -85,B 0,C 180,E1 12582.907,E2 12582.907} C_VEL
LIN {X 0,Y 364.573,Z 723.739,A -85,B 0,C 180,E1 12592.864,E2 12592.864} C_VEL
LIN {X 0,Y 373.581,Z 738.355,A -85,B 0,C 180,E1 12599.297,E2 12599.297} C_VEL
LIN {X 0,Y 388.161,Z 768.161,A -85,B 0,C 180,E1 12606.516,E2 12606.516} C_VEL
LIN {X 0,Y 397.235,Z 800.084,A -85,B 0,C 180,E1 12611.638,E2 12611.638} C_VEL
LIN {X 0,Y 381.228,Z 859.532,A -85,B 0,C 180,E1 12616.646,E2 12616.646} C_VEL
LIN {X 0,Y 363.197,Z 912.759,A -85,B 0,C 180,E1 12624.24,E2 12624.24} C_VEL
LIN {X 0,Y 349.061,Z 953.335,A -85,B 0,C 180,E1 12633.896,E2 12633.896} C_VEL
LIN {X 0,Y 341.209,Z 980.078,A -85,B 0,C 180,E1 12644.672,E2 12644.672} C_VEL
LIN {X 0,Y 339.004,Z 992.556,A -85,B 0,C 180,E1 12654.541,E2 12654.541} C_VEL
LIN {X 0,Y 338.342,Z 994.886,A -85,B 0,C 180,E1 12664.78,E2 12664.78} C_VEL
LIN {X 0,Y 340.11,Z 986.764,A -85,B 0,C 180,E1 12674.805,E2 12674.805} C_VEL
LIN {X 0,Y 345.65,Z 963.99,A -85,B 0,C 180,E1 12686.224,E2 12686.224} C_VEL
LIN {X 0,Y 357.509,Z 927.702,A -85,B 0,C 180,E1 12696.398,E2 12696.398} C_VEL
LIN {X 0,Y 373.545,Z 879.874,A -85,B 0,C 180,E1 12704.56,E2 12704.56} C_VEL
LIN {X 0,Y 390.663,Z 820.025,A -85,B 0,C 180,E1 12710.652,E2 12710.652} C_VEL
LIN {X 0,Y 395.077,Z 793.431,A -85,B 0,C 180,E1 12712.722,E2 12712.722} C_VEL
LIN {X 0,Y 374.94,Z 748.056,A -85,B 0,C 180,E1 12720.492,E2 12720.492} C_VEL
LIN {X 0,Y 350.535,Z 711.158,A -85,B 0,C 180,E1 12729.382,E2 12729.382} C_VEL
LIN {X 0,Y 337.093,Z 691.44,A -85,B 0,C 180,E1 12735.744,E2 12735.744} C_VEL
LIN {X 0,Y 337.282,Z 691.44,A -85,B 0,C 180,E1 12746.347,E2 12746.347} C_VEL
LIN {X 0,Y 337.578,Z 691.44,A -85,B 0,C 180,E1 12757.524,E2 12757.524} C_VEL
LIN {X 0,Y 338.547,Z 691.44,A -85,B 0,C 180,E1 12768.349,E2 12768.349} C_VEL
LIN {X 0,Y 339.42,Z 691.44,A -85,B 0,C 180,E1 12781.263,E2 12781.263} C_VEL
LIN {X 0,Y 338.474,Z 691.44,A -85,B 0,C 180,E1 12791.618,E2 12791.618} C_VEL
LIN {X 0,Y 338.398,Z 693.238,A -85,B 0,C 180,E1 12796.573,E2 12796.573} C_VEL
LIN {X 0,Y 365.135,Z 730.831,A -85,B 0,C 180,E1 12807.093,E2 12807.093} C_VEL
LIN {X 0,Y 391.007,Z 777.239,A -85,B 0,C 180,E1 12815.571,E2 12815.571} C_VEL
LIN {X 0,Y 398.402,Z 799.536,A -85,B 0,C 180,E1 12818.549,E2 12818.549} C_VEL
LIN {X 0,Y 383.082,Z 864.999,A -85,B 0,C 180,E1 12823.164,E2 12823.164} C_VEL
LIN {X 0,Y 366.069,Z 920.918,A -85,B 0,C 180,E1 12830.031,E2 12830.031} C_VEL
LIN {X 0,Y 351.555,Z 965.032,A -85,B 0,C 180,E1 12838.8,E2 12838.8} C_VEL
LIN {X 0,Y 342.429,Z 998.697,A -85,B 0,C 180,E1 12849.911,E2 12849.911} C_VEL
LIN {X 0,Y 339.271,Z 1016.292,A -85,B 0,C 180,E1 12860.992,E2 12860.992} C_VEL
LIN {X 0,Y 339.37,Z 1020.57,A -85,B 0,C 180,E1 12871.281,E2 12871.281} C_VEL
LIN {X 0,Y 339.433,Z 1013.245,A -85,B 0,C 180,E1 12881.606,E2 12881.606} C_VEL
LIN {X 0,Y 343.423,Z 992.939,A -85,B 0,C 180,E1 12892.37,E2 12892.37} C_VEL
LIN {X 0,Y 347.36,Z 978.094,A -85,B 0,C 180,E1 12897.49,E2 12897.49} C_VEL
LIN {X 0,Y 345.342,Z 961.437,A -85,B 0,C 180,E1 12902.665,E2 12902.665} C_VEL
LIN {X 0,Y 362.385,Z 912.521,A -85,B 0,C 180,E1 12912.07,E2 12912.07} C_VEL
LIN {X 0,Y 380.938,Z 854.783,A -85,B 0,C 180,E1 12918.684,E2 12918.684} C_VEL
LIN {X 0,Y 393.933,Z 798.513,A -85,B 0,C 180,E1 12922.718,E2 12922.718} C_VEL
LIN {X 0,Y 378.008,Z 759.153,A -85,B 0,C 180,E1 12930.086,E2 12930.086} C_VEL
LIN {X 0,Y 365.03,Z 736.483,A -85,B 0,C 180,E1 12937.731,E2 12937.731} C_VEL
LIN {X 0,Y 360.415,Z 729.48,A -85,B 0,C 180,E1 12943.241,E2 12943.241} C_VEL
LIN {X 0,Y 362.923,Z 731.88,A -85,B 0,C 180,E1 12952.78,E2 12952.78} C_VEL
LIN {X 0,Y 371.073,Z 745.934,A -85,B 0,C 180,E1 12959.075,E2 12959.075} C_VEL
LIN {X 0,Y 384.868,Z 776.482,A -85,B 0,C 180,E1 12966.523,E2 12966.523} C_VEL
LIN {X 0,Y 391.54,Z 803.57,A -85,B 0,C 180,E1 12970.91,E2 12970.91} C_VEL
LIN {X 0,Y 375.132,Z 861.355,A -85,B 0,C 180,E1 12975.915,E2 12975.915} C_VEL
LIN {X 0,Y 356.255,Z 914.442,A -85,B 0,C 180,E1 12983.672,E2 12983.672} C_VEL
LIN {X 0,Y 341.188,Z 955.439,A -85,B 0,C 180,E1 12993.787,E2 12993.787} C_VEL
LIN {X 0,Y 333.14,Z 981.512,A -85,B 0,C 180,E1 13004.922,E2 13004.922} C_VEL
LIN {X 0,Y 330.916,Z 993.281,A -85,B 0,C 180,E1 13015.023,E2 13015.023} C_VEL
LIN {X 0,Y 330.235,Z 995.353,A -85,B 0,C 180,E1 13024.115,E2 13024.115} C_VEL
LIN {X 0,Y 332.032,Z 987.785,A -85,B 0,C 180,E1 13034.504,E2 13034.504} C_VEL
LIN {X 0,Y 337.628,Z 965.942,A -85,B 0,C 180,E1 13046.135,E2 13046.135} C_VEL
LIN {X 0,Y 349.735,Z 930.684,A -85,B 0,C 180,E1 13056.541,E2 13056.541} C_VEL
LIN {X 0,Y 366.769,Z 882.048,A -85,B 0,C 180,E1 13065.141,E2 13065.141} C_VEL
LIN {X 0,Y 383.981,Z 825.015,A -85,B 0,C 180,E1 13071.14,E2 13071.14} C_VEL
LIN {X 0,Y 389.278,Z 797.203,A -85,B 0,C 180,E1 13073.354,E2 13073.354} C_VEL
LIN {X 0,Y 369.922,Z 752.483,A -85,B 0,C 180,E1 13081.327,E2 13081.327} C_VEL
LIN {X 0,Y 344.782,Z 713.097,A -85,B 0,C 180,E1 13091.204,E2 13091.204} C_VEL
LIN {X 0,Y 329.052,Z 691.44,A -85,B 0,C 180,E1 13099.552,E2 13099.552} C_VEL
LIN {X 0,Y 329.357,Z 691.44,A -85,B 0,C 180,E1 13111.056,E2 13111.056} C_VEL
LIN {X 0,Y 330.011,Z 691.44,A -85,B 0,C 180,E1 13122.596,E2 13122.596} C_VEL
LIN {X 0,Y 330.795,Z 691.44,A -85,B 0,C 180,E1 13133.398,E2 13133.398} C_VEL
LIN {X 0,Y 330.904,Z 691.44,A -85,B 0,C 180,E1 13143.925,E2 13143.925} C_VEL
LIN {X 0,Y 330.478,Z 693.198,A -85,B 0,C 180,E1 13153.082,E2 13153.082} C_VEL
LIN {X 0,Y 352.955,Z 724.188,A -85,B 0,C 180,E1 13163.325,E2 13163.325} C_VEL
LIN {X 0,Y 378.51,Z 766.218,A -85,B 0,C 180,E1 13172.313,E2 13172.313} C_VEL
LIN {X 0,Y 392.644,Z 802.05,A -85,B 0,C 180,E1 13177.799,E2 13177.799} C_VEL
LIN {X 0,Y 377.033,Z 865.807,A -85,B 0,C 180,E1 13182.388,E2 13182.388} C_VEL
LIN {X 0,Y 359.232,Z 921.725,A -85,B 0,C 180,E1 13189.376,E2 13189.376} C_VEL
LIN {X 0,Y 343.977,Z 965.877,A -85,B 0,C 180,E1 13198.404,E2 13198.404} C_VEL
LIN {X 0,Y 334.567,Z 998.703,A -85,B 0,C 180,E1 13209.586,E2 13209.586} C_VEL
LIN {X 0,Y 331.304,Z 1015.989,A -85,B 0,C 180,E1 13220.774,E2 13220.774} C_VEL
LIN {X 0,Y 331.365,Z 1020.27,A -85,B 0,C 180,E1 13231.312,E2 13231.312} C_VEL
LIN {X 0,Y 331.49,Z 1012.931,A -85,B 0,C 180,E1 13241.888,E2 13241.888} C_VEL
LIN {X 0,Y 336.105,Z 991.728,A -85,B 0,C 180,E1 13253.271,E2 13253.271} C_VEL
LIN {X 0,Y 345.342,Z 961.437,A -85,B 0,C 180,E1 13262.665,E2 13262.665} C_VEL
LIN {X 0,Y 345.085,Z 942.511,A -85,B 0,C 180,E1 13267.668,E2 13267.668} C_VEL
LIN {X 0,Y 364.558,Z 888.86,A -85,B 0,C 180,E1 13276.111,E2 13276.111} C_VEL
LIN {X 0,Y 383.541,Z 825.803,A -85,B 0,C 180,E1 13281.893,E2 13281.893} C_VEL
LIN {X 0,Y 388.473,Z 802.135,A -85,B 0,C 180,E1 13283.461,E2 13283.461} C_VEL
LIN {X 0,Y 373.818,Z 764.196,A -85,B 0,C 180,E1 13290.975,E2 13290.975} C_VEL
LIN {X 0,Y 362.54,Z 743.524,A -85,B 0,C 180,E1 13298.378,E2 13298.378} C_VEL
LIN {X 0,Y 358.505,Z 736.98,A -85,B 0,C 180,E1 13304.052,E2 13304.052} C_VEL
LIN {X 0,Y 361.224,Z 740.126,A -85,B 0,C 180,E1 13312.797,E2 13312.797} C_VEL
LIN {X 0,Y 369.181,Z 754.649,A -85,B 0,C 180,E1 13319.258,E2 13319.258} C_VEL
LIN {X 0,Y 381.843,Z 786.591,A -85,B 0,C 180,E1 13326.861,E2 13326.861} C_VEL
LIN {X 0,Y 385.765,Z 807.807,A -85,B 0,C 180,E1 13330.209,E2 13330.209} C_VEL
LIN {X 0,Y 367.922,Z 866.632,A -85,B 0,C 180,E1 13335.563,E2 13335.563} C_VEL
LIN {X 0,Y 348.62,Z 917.86,A -85,B 0,C 180,E1 13343.439,E2 13343.439} C_VEL
LIN {X 0,Y 333.189,Z 957.789,A -85,B 0,C 180,E1 13353.789,E2 13353.789} C_VEL
LIN {X 0,Y 325.086,Z 982.884,A -85,B 0,C 180,E1 13365.141,E2 13365.141} C_VEL
LIN {X 0,Y 322.834,Z 993.9,A -85,B 0,C 180,E1 13375.353,E2 13375.353} C_VEL
LIN {X 0,Y 322.488,Z 994.839,A -85,B 0,C 180,E1 13386.583,E2 13386.583} C_VEL
LIN {X 0,Y 325.098,Z 983.925,A -85,B 0,C 180,E1 13397.874,E2 13397.874} C_VEL
LIN {X 0,Y 332.203,Z 959.167,A -85,B 0,C 180,E1 13409.346,E2 13409.346} C_VEL
LIN {X 0,Y 346.65,Z 920.256,A -85,B 0,C 180,E1 13419.646,E2 13419.646} C_VEL
LIN {X 0,Y 365.305,Z 869.146,A -85,B 0,C 180,E1 13427.686,E2 13427.686} C_VEL
LIN {X 0,Y 382.56,Z 809.069,A -85,B 0,C 180,E1 13433.285,E2 13433.285} C_VEL
LIN {X 0,Y 382.622,Z 798.291,A -85,B 0,C 180,E1 13434.443,E2 13434.443} C_VEL
LIN {X 0,Y 363.595,Z 754.528,A -85,B 0,C 180,E1 13442.694,E2 13442.694} C_VEL
LIN {X 0,Y 341.045,Z 719.152,A -85,B 0,C 180,E1 13452.177,E2 13452.177} C_VEL
LIN {X 0,Y 324.285,Z 697.875,A -85,B 0,C 180,E1 13461.062,E2 13461.062} C_VEL
LIN {X 0,Y 321.087,Z 691.44,A -85,B 0,C 180,E1 13463.778,E2 13463.778} C_VEL
LIN {X 0,Y 321.461,Z 691.44,A -85,B 0,C 180,E1 13476.331,E2 13476.331} C_VEL
LIN {X 0,Y 322.442,Z 691.44,A -85,B 0,C 180,E1 13487.758,E2 13487.758} C_VEL
LIN {X 0,Y 323.048,Z 691.44,A -85,B 0,C 180,E1 13499.074,E2 13499.074} C_VEL
LIN {X 0,Y 322.821,Z 693.301,A -85,B 0,C 180,E1 13509.049,E2 13509.049} C_VEL
LIN {X 0,Y 340.791,Z 717.9,A -85,B 0,C 180,E1 13518.894,E2 13518.894} C_VEL
LIN {X 0,Y 364.08,Z 753.196,A -85,B 0,C 180,E1 13528.105,E2 13528.105} C_VEL
LIN {X 0,Y 385.444,Z 798.161,A -85,B 0,C 180,E1 13536.182,E2 13536.182} C_VEL
LIN {X 0,Y 386.384,Z 807.45,A -85,B 0,C 180,E1 13537.198,E2 13537.198} C_VEL
LIN {X 0,Y 369.602,Z 870.999,A -85,B 0,C 180,E1 13542.024,E2 13542.024} C_VEL
LIN {X 0,Y 351.481,Z 925.251,A -85,B 0,C 180,E1 13549.149,E2 13549.149} C_VEL
LIN {X 0,Y 335.612,Z 969.198,A -85,B 0,C 180,E1 13558.666,E2 13558.666} C_VEL
LIN {X 0,Y 326.176,Z 1000.796,A -85,B 0,C 180,E1 13570.286,E2 13570.286} C_VEL
LIN {X 0,Y 323.208,Z 1016.928,A -85,B 0,C 180,E1 13581.902,E2 13581.902} C_VEL
LIN {X 0,Y 323.375,Z 1019.969,A -85,B 0,C 180,E1 13591.344,E2 13591.344} C_VEL
LIN {X 0,Y 323.546,Z 1012.619,A -85,B 0,C 180,E1 13602.185,E2 13602.185} C_VEL
LIN {X 0,Y 328.553,Z 991.405,A -85,B 0,C 180,E1 13613.838,E2 13613.838} C_VEL
LIN {X 0,Y 340.961,Z 954.273,A -85,B 0,C 180,E1 13625.073,E2 13625.073} C_VEL
LIN {X 0,Y 345.085,Z 942.511,A -85,B 0,C 180,E1 13627.668,E2 13627.668} C_VEL
LIN {X 0,Y 346.554,Z 921.467,A -85,B 0,C 180,E1 13632.403,E2 13632.403} C_VEL
LIN {X 0,Y 367.137,Z 864.812,A -85,B 0,C 180,E1 13639.651,E2 13639.651} C_VEL
LIN {X 0,Y 382.899,Z 805.159,A -85,B 0,C 180,E1 13644.34,E2 13644.34} C_VEL
LIN {X 0,Y 369.168,Z 767.864,A -85,B 0,C 180,E1 13652.172,E2 13652.172} C_VEL
LIN {X 0,Y 359.153,Z 749.011,A -85,B 0,C 180,E1 13659.946,E2 13659.946} C_VEL
LIN {X 0,Y 356.526,Z 744.416,A -85,B 0,C 180,E1 13665.607,E2 13665.607} C_VEL
LIN {X 0,Y 359.299,Z 748.346,A -85,B 0,C 180,E1 13672.878,E2 13672.878} C_VEL
LIN {X 0,Y 366.748,Z 763.046,A -85,B 0,C 180,E1 13679.35,E2 13679.35} C_VEL
LIN {X 0,Y 378.417,Z 796.849,A -85,B 0,C 180,E1 13687.213,E2 13687.213} C_VEL
LIN {X 0,Y 380.118,Z 811.407,A -85,B 0,C 180,E1 13689.464,E2 13689.464} C_VEL
LIN {X 0,Y 361.179,Z 870.667,A -85,B 0,C 180,E1 13695.041,E2 13695.041} C_VEL
LIN {X 0,Y 340.682,Z 922.117,A -85,B 0,C 180,E1 13703.37,E2 13703.37} C_VEL
LIN {X 0,Y 325.034,Z 960.432,A -85,B 0,C 180,E1 13713.927,E2 13713.927} C_VEL
LIN {X 0,Y 317.143,Z 983.819,A -85,B 0,C 180,E1 13725.096,E2 13725.096} C_VEL
LIN {X 0,Y 315.013,Z 993.722,A -85,B 0,C 180,E1 13734.364,E2 13734.364} C_VEL
LIN {X 0,Y 314.32,Z 995.484,A -85,B 0,C 180,E1 13745.771,E2 13745.771} C_VEL
LIN {X 0,Y 316.59,Z 987.1,A -85,B 0,C 180,E1 13756.133,E2 13756.133} C_VEL
LIN {X 0,Y 323.669,Z 963.139,A -85,B 0,C 180,E1 13768.657,E2 13768.657} C_VEL
LIN {X 0,Y 338.588,Z 924.593,A -85,B 0,C 180,E1 13779.594,E2 13779.594} C_VEL
LIN {X 0,Y 357.561,Z 874.666,A -85,B 0,C 180,E1 13787.922,E2 13787.922} C_VEL
LIN {X 0,Y 375.698,Z 815.738,A -85,B 0,C 180,E1 13793.747,E2 13793.747} C_VEL
LIN {X 0,Y 377.099,Z 802.854,A -85,B 0,C 180,E1 13794.997,E2 13794.997} C_VEL
LIN {X 0,Y 359.223,Z 760.136,A -85,B 0,C 180,E1 13803.317,E2 13803.317} C_VEL
LIN {X 0,Y 337.776,Z 725.337,A -85,B 0,C 180,E1 13812.963,E2 13812.963} C_VEL
LIN {X 0,Y 321.783,Z 704.747,A -85,B 0,C 180,E1 13821.913,E2 13821.913} C_VEL
LIN {X 0,Y 315.991,Z 697.608,A -85,B 0,C 180,E1 13826.306,E2 13826.306} C_VEL
LIN {X 0,Y 313.159,Z 691.44,A -85,B 0,C 180,E1 13829.404,E2 13829.404} C_VEL
LIN {X 0,Y 313.827,Z 691.44,A -85,B 0,C 180,E1 13841.667,E2 13841.667} C_VEL
LIN {X 0,Y 314.731,Z 691.44,A -85,B 0,C 180,E1 13853.06,E2 13853.06} C_VEL
LIN {X 0,Y 315.1,Z 693.262,A -85,B 0,C 180,E1 13863.863,E2 13863.863} C_VEL
LIN {X 0,Y 327.295,Z 709.951,A -85,B 0,C 180,E1 13872.7,E2 13872.7} C_VEL
LIN {X 0,Y 347.539,Z 738.25,A -85,B 0,C 180,E1 13882.436,E2 13882.436} C_VEL
LIN {X 0,Y 370.538,Z 779.608,A -85,B 0,C 180,E1 13891.62,E2 13891.62} C_VEL
LIN {X 0,Y 380.982,Z 808.641,A -85,B 0,C 180,E1 13896.335,E2 13896.335} C_VEL
LIN {X 0,Y 363.406,Z 872.385,A -85,B 0,C 180,E1 13901.263,E2 13901.263} C_VEL
LIN {X 0,Y 344.261,Z 927.068,A -85,B 0,C 180,E1 13908.65,E2 13908.65} C_VEL
LIN {X 0,Y 327.684,Z 971.088,A -85,B 0,C 180,E1 13918.561,E2 13918.561} C_VEL
LIN {X 0,Y 318.042,Z 1001.834,A -85,B 0,C 180,E1 13930.487,E2 13930.487} C_VEL
LIN {X 0,Y 315.23,Z 1016.621,A -85,B 0,C 180,E1 13941.695,E2 13941.695} C_VEL
LIN {X 0,Y 315.368,Z 1019.669,A -85,B 0,C 180,E1 13951.378,E2 13951.378} C_VEL
LIN {X 0,Y 315.627,Z 1012.311,A -85,B 0,C 180,E1 13962.495,E2 13962.495} C_VEL
LIN {X 0,Y 321.022,Z 991.097,A -85,B 0,C 180,E1 13974.433,E2 13974.433} C_VEL
LIN {X 0,Y 333.733,Z 955.003,A -85,B 0,C 180,E1 13985.65,E2 13985.65} C_VEL
LIN {X 0,Y 346.554,Z 921.467,A -85,B 0,C 180,E1 13992.403,E2 13992.403} C_VEL
LIN {X 0,Y 349.583,Z 898.321,A -85,B 0,C 180,E1 13996.8,E2 13996.8} C_VEL
LIN {X 0,Y 370.878,Z 836.476,A -85,B 0,C 180,E1 14003.112,E2 14003.112} C_VEL
LIN {X 0,Y 377.643,Z 809.066,A -85,B 0,C 180,E1 14005.098,E2 14005.098} C_VEL
LIN {X 0,Y 365.265,Z 773.593,A -85,B 0,C 180,E1 14012.948,E2 14012.948} C_VEL
LIN {X 0,Y 356.342,Z 754.627,A -85,B 0,C 180,E1 14021.236,E2 14021.236} C_VEL
LIN {X 0,Y 356.505,Z 753.401,A -85,B 0,C 180,E1 14031.452,E2 14031.452} C_VEL
LIN {X 0,Y 363.445,Z 769.511,A -85,B 0,C 180,E1 14038.82,E2 14038.82} C_VEL
LIN {X 0,Y 373.597,Z 802.367,A -85,B 0,C 180,E1 14046.72,E2 14046.72} C_VEL
LIN {X 0,Y 374.509,Z 815.225,A -85,B 0,C 180,E1 14048.706,E2 14048.706} C_VEL
LIN {X 0,Y 355.424,Z 872.04,A -85,B 0,C 180,E1 14054.182,E2 14054.182} C_VEL
LIN {X 0,Y 333.793,Z 923.785,A -85,B 0,C 180,E1 14062.745,E2 14062.745} C_VEL
LIN {X 0,Y 317.653,Z 961.104,A -85,B 0,C 180,E1 14073.336,E2 14073.336} C_VEL
LIN {X 0,Y 309.358,Z 984.159,A -85,B 0,C 180,E1 14084.659,E2 14084.659} C_VEL
LIN {X 0,Y 306.776,Z 994.714,A -85,B 0,C 180,E1 14095.328,E2 14095.328} C_VEL
LIN {X 0,Y 306.379,Z 995.581,A -85,B 0,C 180,E1 14106.401,E2 14106.401} C_VEL
LIN {X 0,Y 308.914,Z 986.404,A -85,B 0,C 180,E1 14117.229,E2 14117.229} C_VEL
LIN {X 0,Y 316.248,Z 963.391,A -85,B 0,C 180,E1 14129.313,E2 14129.313} C_VEL
LIN {X 0,Y 331.463,Z 926.054,A -85,B 0,C 180,E1 14140.157,E2 14140.157} C_VEL
LIN {X 0,Y 350.593,Z 877.953,A -85,B 0,C 180,E1 14148.454,E2 14148.454} C_VEL
LIN {X 0,Y 369.668,Z 819.237,A -85,B 0,C 180,E1 14154.462,E2 14154.462} C_VEL
LIN {X 0,Y 371.407,Z 806.79,A -85,B 0,C 180,E1 14155.665,E2 14155.665} C_VEL
LIN {X 0,Y 354.254,Z 764.301,A -85,B 0,C 180,E1 14164.255,E2 14164.255} C_VEL
LIN {X 0,Y 332.483,Z 728.133,A -85,B 0,C 180,E1 14174.828,E2 14174.828} C_VEL
LIN {X 0,Y 315.744,Z 706.212,A -85,B 0,C 180,E1 14185.614,E2 14185.614} C_VEL
LIN {X 0,Y 308.976,Z 698.173,A -85,B 0,C 180,E1 14192.442,E2 14192.442} C_VEL
LIN {X 0,Y 305.753,Z 691.44,A -85,B 0,C 180,E1 14201.165,E2 14201.165} C_VEL
LIN {X 0,Y 306.734,Z 691.44,A -85,B 0,C 180,E1 14212.878,E2 14212.878} C_VEL
LIN {X 0,Y 313.879,Z 702.14,A -85,B 0,C 180,E1 14223.878,E2 14223.878} C_VEL
LIN {X 0,Y 325.293,Z 717.158,A -85,B 0,C 180,E1 14232.215,E2 14232.215} C_VEL
LIN {X 0,Y 346.097,Z 747.205,A -85,B 0,C 180,E1 14242.62,E2 14242.62} C_VEL
LIN {X 0,Y 367.876,Z 789.616,A -85,B 0,C 180,E1 14251.93,E2 14251.93} C_VEL
LIN {X 0,Y 374.897,Z 813.014,A -85,B 0,C 180,E1 14255.642,E2 14255.642} C_VEL
LIN {X 0,Y 356.101,Z 877.32,A -85,B 0,C 180,E1 14260.847,E2 14260.847} C_VEL
LIN {X 0,Y 335.866,Z 931.903,A -85,B 0,C 180,E1 14268.672,E2 14268.672} C_VEL
LIN {X 0,Y 319.334,Z 973.99,A -85,B 0,C 180,E1 14278.822,E2 14278.822} C_VEL
LIN {X 0,Y 309.891,Z 1002.819,A -85,B 0,C 180,E1 14290.697,E2 14290.697} C_VEL
LIN {X 0,Y 307.194,Z 1017.231,A -85,B 0,C 180,E1 14302.905,E2 14302.905} C_VEL
LIN {X 0,Y 307.169,Z 1018.619,A -85,B 0,C 180,E1 14314.249,E2 14314.249} C_VEL
LIN {X 0,Y 308.656,Z 1008.315,A -85,B 0,C 180,E1 14325.689,E2 14325.689} C_VEL
LIN {X 0,Y 315.68,Z 983.475,A -85,B 0,C 180,E1 14337.95,E2 14337.95} C_VEL
LIN {X 0,Y 331.433,Z 943.317,A -85,B 0,C 180,E1 14349.158,E2 14349.158} C_VEL
LIN {X 0,Y 349.583,Z 898.321,A -85,B 0,C 180,E1 14356.8,E2 14356.8} C_VEL
LIN {X 0,Y 353.791,Z 873.095,A -85,B 0,C 180,E1 14360.816,E2 14360.816} C_VEL
LIN {X 0,Y 372.372,Z 813.116,A -85,B 0,C 180,E1 14365.835,E2 14365.835} C_VEL
LIN {X 0,Y 361.899,Z 780.315,A -85,B 0,C 180,E1 14373.375,E2 14373.375} C_VEL
LIN {X 0,Y 353.999,Z 761.256,A -85,B 0,C 180,E1 14381.916,E2 14381.916} C_VEL
LIN {X 0,Y 354.358,Z 762.325,A -85,B 0,C 180,E1 14391.864,E2 14391.864} C_VEL
LIN {X 0,Y 360.451,Z 777.61,A -85,B 0,C 180,E1 14398.811,E2 14398.811} C_VEL
LIN {X 0,Y 369.111,Z 809.38,A -85,B 0,C 180,E1 14406.506,E2 14406.506} C_VEL
LIN {X 0,Y 368.66,Z 820.13,A -85,B 0,C 180,E1 14407.999,E2 14407.999} C_VEL
LIN {X 0,Y 347.768,Z 878.068,A -85,B 0,C 180,E1 14413.9,E2 14413.9} C_VEL
LIN {X 0,Y 326.15,Z 926.968,A -85,B 0,C 180,E1 14422.444,E2 14422.444} C_VEL
LIN {X 0,Y 309.282,Z 964.328,A -85,B 0,C 180,E1 14433.688,E2 14433.688} C_VEL
LIN {X 0,Y 301.126,Z 986.273,A -85,B 0,C 180,E1 14445.528,E2 14445.528} C_VEL
LIN {X 0,Y 298.387,Z 995.897,A -85,B 0,C 180,E1 14457.059,E2 14457.059} C_VEL
LIN {X 0,Y 298.525,Z 995.495,A -85,B 0,C 180,E1 14467.588,E2 14467.588} C_VEL
LIN {X 0,Y 301.474,Z 984.923,A -85,B 0,C 180,E1 14478.993,E2 14478.993} C_VEL
LIN {X 0,Y 310.208,Z 959.92,A -85,B 0,C 180,E1 14491.402,E2 14491.402} C_VEL
LIN {X 0,Y 326.766,Z 921.692,A -85,B 0,C 180,E1 14502.064,E2 14502.064} C_VEL
LIN {X 0,Y 347.905,Z 870.291,A -85,B 0,C 180,E1 14510.426,E2 14510.426} C_VEL
LIN {X 0,Y 365.777,Z 811.197,A -85,B 0,C 180,E1 14516.239,E2 14516.239} C_VEL
LIN {X 0,Y 350.419,Z 771.121,A -85,B 0,C 180,E1 14524.582,E2 14524.582} C_VEL
LIN {X 0,Y 330.115,Z 735.57,A -85,B 0,C 180,E1 14535.137,E2 14535.137} C_VEL
LIN {X 0,Y 314.036,Z 713.806,A -85,B 0,C 180,E1 14546.036,E2 14546.036} C_VEL
LIN {X 0,Y 306.992,Z 705.453,A -85,B 0,C 180,E1 14553.571,E2 14553.571} C_VEL
LIN {X 0,Y 303.709,Z 699.166,A -85,B 0,C 180,E1 14561.033,E2 14561.033} C_VEL
LIN {X 0,Y 305.89,Z 701.419,A -85,B 0,C 180,E1 14575.447,E2 14575.447} C_VEL
LIN {X 0,Y 312.62,Z 710.318,A -85,B 0,C 180,E1 14583.785,E2 14583.785} C_VEL
LIN {X 0,Y 323.919,Z 725.587,A -85,B 0,C 180,E1 14592.208,E2 14592.208} C_VEL
LIN {X 0,Y 343.642,Z 755.482,A -85,B 0,C 180,E1 14602.516,E2 14602.516} C_VEL
LIN {X 0,Y 364.076,Z 797.405,A -85,B 0,C 180,E1 14611.836,E2 14611.836} C_VEL
LIN {X 0,Y 369.194,Z 815.708,A -85,B 0,C 180,E1 14614.839,E2 14614.839} C_VEL
LIN {X 0,Y 350.223,Z 877.916,A -85,B 0,C 180,E1 14619.964,E2 14619.964} C_VEL
LIN {X 0,Y 328.952,Z 933.017,A -85,B 0,C 180,E1 14628.014,E2 14628.014} C_VEL
LIN {X 0,Y 311.339,Z 975.833,A -85,B 0,C 180,E1 14638.753,E2 14638.753} C_VEL
LIN {X 0,Y 301.729,Z 1003.662,A -85,B 0,C 180,E1 14650.917,E2 14650.917} C_VEL
LIN {X 0,Y 299.196,Z 1016.923,A -85,B 0,C 180,E1 14662.714,E2 14662.714} C_VEL
LIN {X 0,Y 299.354,Z 1019.068,A -85,B 0,C 180,E1 14671.452,E2 14671.452} C_VEL
LIN {X 0,Y 299.781,Z 1011.704,A -85,B 0,C 180,E1 14683.167,E2 14683.167} C_VEL
LIN {X 0,Y 305.88,Z 990.724,A -85,B 0,C 180,E1 14695.623,E2 14695.623} C_VEL
LIN {X 0,Y 320.513,Z 953.854,A -85,B 0,C 180,E1 14707.561,E2 14707.561} C_VEL
LIN {X 0,Y 340.879,Z 905.638,A -85,B 0,C 180,E1 14716.763,E2 14716.763} C_VEL
LIN {X 0,Y 353.791,Z 873.095,A -85,B 0,C 180,E1 14720.816,E2 14720.816} C_VEL
LIN {X 0,Y 358.494,Z 846.024,A -85,B 0,C 180,E1 14724.433,E2 14724.433} C_VEL
LIN {X 0,Y 366.863,Z 815.619,A -85,B 0,C 180,E1 14726.896,E2 14726.896} C_VEL
LIN {X 0,Y 357.217,Z 783.529,A -85,B 0,C 180,E1 14734.889,E2 14734.889} C_VEL
LIN {X 0,Y 351.195,Z 768.507,A -85,B 0,C 180,E1 14742.742,E2 14742.742} C_VEL
LIN {X 0,Y 351.957,Z 770.339,A -85,B 0,C 180,E1 14751.886,E2 14751.886} C_VEL
LIN {X 0,Y 357.748,Z 786.545,A -85,B 0,C 180,E1 14759.137,E2 14759.137} C_VEL
LIN {X 0,Y 364.676,Z 818.116,A -85,B 0,C 180,E1 14766.672,E2 14766.672} C_VEL
LIN {X 0,Y 343.737,Z 875.757,A -85,B 0,C 180,E1 14772.497,E2 14772.497} C_VEL
LIN {X 0,Y 320.937,Z 925.417,A -85,B 0,C 180,E1 14781.03,E2 14781.03} C_VEL
LIN {X 0,Y 302.324,Z 964.076,A -85,B 0,C 180,E1 14792.689,E2 14792.689} C_VEL
LIN {X 0,Y 293.598,Z 985.627,A -85,B 0,C 180,E1 14804.26,E2 14804.26} C_VEL
LIN {X 0,Y 291.071,Z 994.776,A -85,B 0,C 180,E1 14813.921,E2 14813.921} C_VEL
LIN {X 0,Y 290.368,Z 996.069,A -85,B 0,C 180,E1 14826.923,E2 14826.923} C_VEL
LIN {X 0,Y 293.415,Z 986.141,A -85,B 0,C 180,E1 14838.687,E2 14838.687} C_VEL
LIN {X 0,Y 302.217,Z 962.013,A -85,B 0,C 180,E1 14851.439,E2 14851.439} C_VEL
LIN {X 0,Y 319.089,Z 924.778,A -85,B 0,C 180,E1 14862.359,E2 14862.359} C_VEL
LIN {X 0,Y 340.547,Z 874.994,A -85,B 0,C 180,E1 14870.827,E2 14870.827} C_VEL
LIN {X 0,Y 360.131,Z 815.349,A -85,B 0,C 180,E1 14876.877,E2 14876.877} C_VEL
LIN {X 0,Y 345.822,Z 776.425,A -85,B 0,C 180,E1 14885.284,E2 14885.284} C_VEL
LIN {X 0,Y 326.902,Z 742.27,A -85,B 0,C 180,E1 14895.811,E2 14895.811} C_VEL
LIN {X 0,Y 312.029,Z 721.223,A -85,B 0,C 180,E1 14906.61,E2 14906.61} C_VEL
LIN {X 0,Y 305.554,Z 713.102,A -85,B 0,C 180,E1 14914.042,E2 14914.042} C_VEL
LIN {X 0,Y 302.27,Z 706.982,A -85,B 0,C 180,E1 14922.444,E2 14922.444} C_VEL
LIN {X 0,Y 304.652,Z 709.239,A -85,B 0,C 180,E1 14935.202,E2 14935.202} C_VEL
LIN {X 0,Y 311.386,Z 718.53,A -85,B 0,C 180,E1 14943.735,E2 14943.735} C_VEL
LIN {X 0,Y 324.788,Z 736.618,A -85,B 0,C 180,E1 14953.592,E2 14953.592} C_VEL
LIN {X 0,Y 345.024,Z 770.888,A -85,B 0,C 180,E1 14964.367,E2 14964.367} C_VEL
LIN {X 0,Y 362.808,Z 813.27,A -85,B 0,C 180,E1 14973.266,E2 14973.266} C_VEL
LIN {X 0,Y 362.164,Z 823.964,A -85,B 0,C 180,E1 14974.366,E2 14974.366} C_VEL
LIN {X 0,Y 341.44,Z 886.56,A -85,B 0,C 180,E1 14980,E2 14980} C_VEL
LIN {X 0,Y 320.524,Z 937.474,A -85,B 0,C 180,E1 14988.026,E2 14988.026} C_VEL
LIN {X 0,Y 303.279,Z 977.757,A -85,B 0,C 180,E1 14998.723,E2 14998.723} C_VEL
LIN {X 0,Y 293.18,Z 1005.687,A -85,B 0,C 180,E1 15011.905,E2 15011.905} C_VEL
LIN {X 0,Y 291.211,Z 1016.612,A -85,B 0,C 180,E1 15022.513,E2 15022.513} C_VEL
LIN {X 0,Y 291.353,Z 1018.768,A -85,B 0,C 180,E1 15031.492,E2 15031.492} C_VEL
LIN {X 0,Y 291.871,Z 1011.407,A -85,B 0,C 180,E1 15043.531,E2 15043.531} C_VEL
LIN {X 0,Y 298.622,Z 989.778,A -85,B 0,C 180,E1 15056.601,E2 15056.601} C_VEL
LIN {X 0,Y 314.298,Z 952.589,A -85,B 0,C 180,E1 15068.773,E2 15068.773} C_VEL
LIN {X 0,Y 336.282,Z 903.261,A -85,B 0,C 180,E1 15078.126,E2 15078.126} C_VEL
LIN {X 0,Y 358.494,Z 846.024,A -85,B 0,C 180,E1 15084.433,E2 15084.433} C_VEL
LIN {X 0,Y 362.03,Z 821.311,A -85,B 0,C 180,E1 15087.399,E2 15087.399} C_VEL
LIN {X 0,Y 361.562,Z 818.458,A -85,B 0,C 180,E1 15087.94,E2 15087.94} C_VEL
LIN {X 0,Y 353.195,Z 788.713,A -85,B 0,C 180,E1 15095.936,E2 15095.936} C_VEL
LIN {X 0,Y 348.439,Z 775.762,A -85,B 0,C 180,E1 15103.578,E2 15103.578} C_VEL
LIN {X 0,Y 349.139,Z 776.997,A -85,B 0,C 180,E1 15111.27,E2 15111.27} C_VEL
LIN {X 0,Y 354.115,Z 793.328,A -85,B 0,C 180,E1 15118.789,E2 15118.789} C_VEL
LIN {X 0,Y 359.553,Z 822.298,A -85,B 0,C 180,E1 15125.92,E2 15125.92} C_VEL
LIN {X 0,Y 337.006,Z 879.987,A -85,B 0,C 180,E1 15131.928,E2 15131.928} C_VEL
LIN {X 0,Y 313.589,Z 928.231,A -85,B 0,C 180,E1 15140.605,E2 15140.605} C_VEL
LIN {X 0,Y 295.118,Z 964.611,A -85,B 0,C 180,E1 15151.954,E2 15151.954} C_VEL
LIN {X 0,Y 285.308,Z 987.594,A -85,B 0,C 180,E1 15165.125,E2 15165.125} C_VEL
LIN {X 0,Y 282.498,Z 996.396,A -85,B 0,C 180,E1 15176.381,E2 15176.381} C_VEL
LIN {X 0,Y 282.852,Z 995.143,A -85,B 0,C 180,E1 15189.59,E2 15189.59} C_VEL
LIN {X 0,Y 286.462,Z 982.982,A -85,B 0,C 180,E1 15201.649,E2 15201.649} C_VEL
LIN {X 0,Y 297.578,Z 956.511,A -85,B 0,C 180,E1 15214.388,E2 15214.388} C_VEL
LIN {X 0,Y 317.027,Z 915.829,A -85,B 0,C 180,E1 15225.266,E2 15225.266} C_VEL
LIN {X 0,Y 339.619,Z 863.57,A -85,B 0,C 180,E1 15233.274,E2 15233.274} C_VEL
LIN {X 0,Y 354.15,Z 818.316,A -85,B 0,C 180,E1 15237.769,E2 15237.769} C_VEL
LIN {X 0,Y 340.339,Z 779.833,A -85,B 0,C 180,E1 15246.5,E2 15246.5} C_VEL
LIN {X 0,Y 323.151,Z 748.321,A -85,B 0,C 180,E1 15256.774,E2 15256.774} C_VEL
LIN {X 0,Y 309.844,Z 728.489,A -85,B 0,C 180,E1 15267.286,E2 15267.286} C_VEL
LIN {X 0,Y 303.626,Z 720.405,A -85,B 0,C 180,E1 15275.044,E2 15275.044} C_VEL
LIN {X 0,Y 301.17,Z 714.897,A -85,B 0,C 180,E1 15282.378,E2 15282.378} C_VEL
LIN {X 0,Y 303.44,Z 717.185,A -85,B 0,C 180,E1 15295.058,E2 15295.058} C_VEL
LIN {X 0,Y 309.979,Z 726.62,A -85,B 0,C 180,E1 15303.664,E2 15303.664} C_VEL
LIN {X 0,Y 322.883,Z 745.153,A -85,B 0,C 180,E1 15313.565,E2 15313.565} C_VEL
LIN {X 0,Y 341.51,Z 777.884,A -85,B 0,C 180,E1 15324.021,E2 15324.021} C_VEL
LIN {X 0,Y 357.995,Z 819.866,A -85,B 0,C 180,E1 15333.026,E2 15333.026} C_VEL
LIN {X 0,Y 337.567,Z 881.933,A -85,B 0,C 180,E1 15338.452,E2 15338.452} C_VEL
LIN {X 0,Y 315.895,Z 933.619,A -85,B 0,C 180,E1 15346.322,E2 15346.322} C_VEL
LIN {X 0,Y 296.469,Z 976.427,A -85,B 0,C 180,E1 15357.561,E2 15357.561} C_VEL
LIN {X 0,Y 285.824,Z 1004.152,A -85,B 0,C 180,E1 15370.618,E2 15370.618} C_VEL
LIN {X 0,Y 283.215,Z 1016.298,A -85,B 0,C 180,E1 15382.301,E2 15382.301} C_VEL
LIN {X 0,Y 283.345,Z 1018.468,A -85,B 0,C 180,E1 15391.534,E2 15391.534} C_VEL
LIN {X 0,Y 284.003,Z 1011.114,A -85,B 0,C 180,E1 15403.913,E2 15403.913} C_VEL
LIN {X 0,Y 291.141,Z 989.506,A -85,B 0,C 180,E1 15417.34,E2 15417.34} C_VEL
LIN {X 0,Y 308.27,Z 951.421,A -85,B 0,C 180,E1 15430.007,E2 15430.007} C_VEL
LIN {X 0,Y 331.549,Z 901.777,A -85,B 0,C 180,E1 15439.398,E2 15439.398} C_VEL
LIN {X 0,Y 355.165,Z 842.494,A -85,B 0,C 180,E1 15445.826,E2 15445.826} C_VEL
LIN {X 0,Y 361.857,Z 819.902,A -85,B 0,C 180,E1 15447.65,E2 15447.65} C_VEL
LIN {X 0,Y 361.562,Z 818.458,A -85,B 0,C 180,E1 15447.94,E2 15447.94} C_VEL
LIN {X 0,Y 352.627,Z 805.334,A -85,B 0,C 180,E1 15453.072,E2 15453.072} C_VEL
LIN {X 0,Y 346.725,Z 786.654,A -85,B 0,C 180,E1 15460.861,E2 15460.861} C_VEL
LIN {X 0,Y 345.514,Z 782.887,A -85,B 0,C 180,E1 15468.622,E2 15468.622} C_VEL
LIN {X 0,Y 348.512,Z 792.289,A -85,B 0,C 180,E1 15475.568,E2 15475.568} C_VEL
LIN {X 0,Y 353.478,Z 817.787,A -85,B 0,C 180,E1 15483.246,E2 15483.246} C_VEL
LIN {X 0,Y 353.599,Z 828.156,A -85,B 0,C 180,E1 15485.248,E2 15485.248} C_VEL
LIN {X 0,Y 329.767,Z 885.354,A -85,B 0,C 180,E1 15491.481,E2 15491.481} C_VEL
LIN {X 0,Y 304.34,Z 934.486,A -85,B 0,C 180,E1 15500.98,E2 15500.98} C_VEL
LIN {X 0,Y 285.499,Z 969.937,A -85,B 0,C 180,E1 15513.365,E2 15513.365} C_VEL
LIN {X 0,Y 276.891,Z 990.251,A -85,B 0,C 180,E1 15526.757,E2 15526.757} C_VEL
LIN {X 0,Y 274.123,Z 997.505,A -85,B 0,C 180,E1 15539.113,E2 15539.113} C_VEL
LIN {X 0,Y 275.487,Z 993.792,A -85,B 0,C 180,E1 15552.364,E2 15552.364} C_VEL
LIN {X 0,Y 281.439,Z 977.143,A -85,B 0,C 180,E1 15566.011,E2 15566.011} C_VEL
LIN {X 0,Y 296.455,Z 945.653,A -85,B 0,C 180,E1 15578.835,E2 15578.835} C_VEL
LIN {X 0,Y 317.546,Z 902.357,A -85,B 0,C 180,E1 15588.82,E2 15588.82} C_VEL
LIN {X 0,Y 340.565,Z 847.419,A -85,B 0,C 180,E1 15596.107,E2 15596.107} C_VEL
LIN {X 0,Y 348.398,Z 822.141,A -85,B 0,C 180,E1 15598.512,E2 15598.512} C_VEL
LIN {X 0,Y 335.916,Z 785.614,A -85,B 0,C 180,E1 15607.077,E2 15607.077} C_VEL
LIN {X 0,Y 320.006,Z 754.98,A -85,B 0,C 180,E1 15617.392,E2 15617.392} C_VEL
LIN {X 0,Y 307.698,Z 735.915,A -85,B 0,C 180,E1 15627.763,E2 15627.763} C_VEL
LIN {X 0,Y 301.87,Z 727.685,A -85,B 0,C 180,E1 15635.879,E2 15635.879} C_VEL
LIN {X 0,Y 299.688,Z 722.651,A -85,B 0,C 180,E1 15643.814,E2 15643.814} C_VEL
LIN {X 0,Y 302.122,Z 725.276,A -85,B 0,C 180,E1 15655.037,E2 15655.037} C_VEL
LIN {X 0,Y 308.557,Z 734.724,A -85,B 0,C 180,E1 15663.681,E2 15663.681} C_VEL
LIN {X 0,Y 321.405,Z 754.461,A -85,B 0,C 180,E1 15673.949,E2 15673.949} C_VEL
LIN {X 0,Y 337.999,Z 785.374,A -85,B 0,C 180,E1 15683.814,E2 15683.814} C_VEL
LIN {X 0,Y 352.216,Z 824.545,A -85,B 0,C 180,E1 15692.346,E2 15692.346} C_VEL
LIN {X 0,Y 330.399,Z 886.327,A -85,B 0,C 180,E1 15697.945,E2 15697.945} C_VEL
LIN {X 0,Y 307.135,Z 938.633,A -85,B 0,C 180,E1 15706.422,E2 15706.422} C_VEL
LIN {X 0,Y 288.505,Z 978.078,A -85,B 0,C 180,E1 15717.449,E2 15717.449} C_VEL
LIN {X 0,Y 277.667,Z 1004.98,A -85,B 0,C 180,E1 15730.856,E2 15730.856} C_VEL
LIN {X 0,Y 275.248,Z 1015.984,A -85,B 0,C 180,E1 15742.077,E2 15742.077} C_VEL
LIN {X 0,Y 275.355,Z 1018.169,A -85,B 0,C 180,E1 15751.578,E2 15751.578} C_VEL
LIN {X 0,Y 276.109,Z 1010.825,A -85,B 0,C 180,E1 15764.319,E2 15764.319} C_VEL
LIN {X 0,Y 283.958,Z 988.49,A -85,B 0,C 180,E1 15778.457,E2 15778.457} C_VEL
LIN {X 0,Y 301.575,Z 951.888,A -85,B 0,C 180,E1 15790.86,E2 15790.86} C_VEL
LIN {X 0,Y 326.151,Z 902.072,A -85,B 0,C 180,E1 15800.459,E2 15800.459} C_VEL
LIN {X 0,Y 350.826,Z 842.696,A -85,B 0,C 180,E1 15806.941,E2 15806.941} C_VEL
LIN {X 0,Y 356.755,Z 823.872,A -85,B 0,C 180,E1 15808.477,E2 15808.477} C_VEL
LIN {X 0,Y 352.627,Z 805.334,A -85,B 0,C 180,E1 15813.072,E2 15813.072} C_VEL
LIN {X 0,Y 344.954,Z 797.895,A -85,B 0,C 180,E1 15818.68,E2 15818.68} C_VEL
LIN {X 0,Y 342.492,Z 790.258,A -85,B 0,C 180,E1 15825.918,E2 15825.918} C_VEL
LIN {X 0,Y 344.451,Z 795.845,A -85,B 0,C 180,E1 15833.696,E2 15833.696} C_VEL
LIN {X 0,Y 348.415,Z 820.091,A -85,B 0,C 180,E1 15841.888,E2 15841.888} C_VEL
LIN {X 0,Y 348.177,Z 832.53,A -85,B 0,C 180,E1 15844.407,E2 15844.407} C_VEL
LIN {X 0,Y 322.911,Z 889.592,A -85,B 0,C 180,E1 15850.897,E2 15850.897} C_VEL
LIN {X 0,Y 297.243,Z 936.701,A -85,B 0,C 180,E1 15860.398,E2 15860.398} C_VEL
LIN {X 0,Y 277.695,Z 971.605,A -85,B 0,C 180,E1 15873.146,E2 15873.146} C_VEL
LIN {X 0,Y 268.999,Z 990.717,A -85,B 0,C 180,E1 15886.425,E2 15886.425} C_VEL
LIN {X 0,Y 266.264,Z 997.379,A -85,B 0,C 180,E1 15897.218,E2 15897.218} C_VEL
LIN {X 0,Y 266.853,Z 995.836,A -85,B 0,C 180,E1 15909.786,E2 15909.786} C_VEL
LIN {X 0,Y 271.011,Z 983.513,A -85,B 0,C 180,E1 15922.763,E2 15922.763} C_VEL
LIN {X 0,Y 283.724,Z 956.78,A -85,B 0,C 180,E1 15936.171,E2 15936.171} C_VEL
LIN {X 0,Y 305.087,Z 915.933,A -85,B 0,C 180,E1 15947.366,E2 15947.366} C_VEL
LIN {X 0,Y 329.305,Z 863.507,A -85,B 0,C 180,E1 15955.46,E2 15955.46} C_VEL
LIN {X 0,Y 342.327,Z 824.679,A -85,B 0,C 180,E1 15959.535,E2 15959.535} C_VEL
LIN {X 0,Y 330.089,Z 788.035,A -85,B 0,C 180,E1 15968.612,E2 15968.612} C_VEL
LIN {X 0,Y 314.576,Z 757.474,A -85,B 0,C 180,E1 15979.739,E2 15979.739} C_VEL
LIN {X 0,Y 302.838,Z 737.968,A -85,B 0,C 180,E1 15991.908,E2 15991.908} C_VEL
LIN {X 0,Y 298.36,Z 730.513,A -85,B 0,C 180,E1 16003.74,E2 16003.74} C_VEL
LIN {X 0,Y 300.609,Z 732.993,A -85,B 0,C 180,E1 16014.761,E2 16014.761} C_VEL
LIN {X 0,Y 306.736,Z 742.495,A -85,B 0,C 180,E1 16023.525,E2 16023.525} C_VEL
LIN {X 0,Y 320.244,Z 763.856,A -85,B 0,C 180,E1 16034.57,E2 16034.57} C_VEL
LIN {X 0,Y 336.621,Z 798.081,A -85,B 0,C 180,E1 16044.973,E2 16044.973} C_VEL
LIN {X 0,Y 346.031,Z 829.137,A -85,B 0,C 180,E1 16051.599,E2 16051.599} C_VEL
LIN {X 0,Y 323.89,Z 888.964,A -85,B 0,C 180,E1 16057.213,E2 16057.213} C_VEL
LIN {X 0,Y 299.518,Z 941.278,A -85,B 0,C 180,E1 16066.016,E2 16066.016} C_VEL
LIN {X 0,Y 279.952,Z 980.803,A -85,B 0,C 180,E1 16077.775,E2 16077.775} C_VEL
LIN {X 0,Y 269.492,Z 1005.76,A -85,B 0,C 180,E1 16091.106,E2 16091.106} C_VEL
LIN {X 0,Y 267.089,Z 1016.568,A -85,B 0,C 180,E1 16103.514,E2 16103.514} C_VEL
LIN {X 0,Y 267.168,Z 1017.131,A -85,B 0,C 180,E1 16114.887,E2 16114.887} C_VEL
LIN {X 0,Y 269.552,Z 1005.832,A -85,B 0,C 180,E1 16128.888,E2 16128.888} C_VEL
LIN {X 0,Y 280.114,Z 980.507,A -85,B 0,C 180,E1 16142.65,E2 16142.65} C_VEL
LIN {X 0,Y 301.073,Z 940.888,A -85,B 0,C 180,E1 16154.577,E2 16154.577} C_VEL
LIN {X 0,Y 327.304,Z 889.101,A -85,B 0,C 180,E1 16163.359,E2 16163.359} C_VEL
LIN {X 0,Y 351.529,Z 826.929,A -85,B 0,C 180,E1 16169.55,E2 16169.55} C_VEL
LIN {X 0,Y 345.768,Z 800.472,A -85,B 0,C 180,E1 16177.443,E2 16177.443} C_VEL
LIN {X 0,Y 344.954,Z 797.895,A -85,B 0,C 180,E1 16178.68,E2 16178.68} C_VEL
LIN {X 0,Y 339.743,Z 798.086,A -85,B 0,C 180,E1 16184.604,E2 16184.604} C_VEL
LIN {X 0,Y 340.507,Z 800.977,A -85,B 0,C 180,E1 16191.972,E2 16191.972} C_VEL
LIN {X 0,Y 343.255,Z 819.842,A -85,B 0,C 180,E1 16199.701,E2 16199.701} C_VEL
LIN {X 0,Y 343.635,Z 835.011,A -85,B 0,C 180,E1 16203.387,E2 16203.387} C_VEL
LIN {X 0,Y 317.662,Z 890.948,A -85,B 0,C 180,E1 16209.838,E2 16209.838} C_VEL
LIN {X 0,Y 290.55,Z 938.291,A -85,B 0,C 180,E1 16219.612,E2 16219.612} C_VEL
LIN {X 0,Y 269.976,Z 972.972,A -85,B 0,C 180,E1 16232.801,E2 16232.801} C_VEL
LIN {X 0,Y 260.952,Z 991.684,A -85,B 0,C 180,E1 16246.643,E2 16246.643} C_VEL
LIN {X 0,Y 257.942,Z 998.214,A -85,B 0,C 180,E1 16259.995,E2 16259.995} C_VEL
LIN {X 0,Y 259.578,Z 994.387,A -85,B 0,C 180,E1 16272.913,E2 16272.913} C_VEL
LIN {X 0,Y 266.67,Z 977.28,A -85,B 0,C 180,E1 16287.608,E2 16287.608} C_VEL
LIN {X 0,Y 283.264,Z 945.922,A -85,B 0,C 180,E1 16300.808,E2 16300.808} C_VEL
LIN {X 0,Y 306.316,Z 902.293,A -85,B 0,C 180,E1 16311.051,E2 16311.051} C_VEL
LIN {X 0,Y 331.161,Z 846.72,A -85,B 0,C 180,E1 16318.389,E2 16318.389} C_VEL
LIN {X 0,Y 336.594,Z 828.468,A -85,B 0,C 180,E1 16320.316,E2 16320.316} C_VEL
LIN {X 0,Y 325.153,Z 792.437,A -85,B 0,C 180,E1 16329.633,E2 16329.633} C_VEL
LIN {X 0,Y 310.944,Z 763.728,A -85,B 0,C 180,E1 16340.645,E2 16340.645} C_VEL
LIN {X 0,Y 300.622,Z 745.54,A -85,B 0,C 180,E1 16352.422,E2 16352.422} C_VEL
LIN {X 0,Y 296.757,Z 738.356,A -85,B 0,C 180,E1 16363.649,E2 16363.649} C_VEL
LIN {X 0,Y 298.901,Z 740.821,A -85,B 0,C 180,E1 16374.618,E2 16374.618} C_VEL
LIN {X 0,Y 305.15,Z 750.849,A -85,B 0,C 180,E1 16383.811,E2 16383.811} C_VEL
LIN {X 0,Y 317.644,Z 772.142,A -85,B 0,C 180,E1 16394.59,E2 16394.59} C_VEL
LIN {X 0,Y 332.397,Z 804.547,A -85,B 0,C 180,E1 16404.592,E2 16404.592} C_VEL
LIN {X 0,Y 340.292,Z 832.584,A -85,B 0,C 180,E1 16410.754,E2 16410.754} C_VEL
LIN {X 0,Y 317.246,Z 891.759,A -85,B 0,C 180,E1 16416.491,E2 16416.491} C_VEL
LIN {X 0,Y 292.168,Z 943.273,A -85,B 0,C 180,E1 16425.474,E2 16425.474} C_VEL
LIN {X 0,Y 271.522,Z 983.061,A -85,B 0,C 180,E1 16437.928,E2 16437.928} C_VEL
LIN {X 0,Y 261.324,Z 1006.397,A -85,B 0,C 180,E1 16451.372,E2 16451.372} C_VEL
LIN {X 0,Y 259.109,Z 1016.819,A -85,B 0,C 180,E1 16464.959,E2 16464.959} C_VEL
LIN {X 0,Y 259.182,Z 1016.838,A -85,B 0,C 180,E1 16475.038,E2 16475.038} C_VEL
LIN {X 0,Y 261.47,Z 1006.576,A -85,B 0,C 180,E1 16488.615,E2 16488.615} C_VEL
LIN {X 0,Y 272.482,Z 981.527,A -85,B 0,C 180,E1 16503.1,E2 16503.1} C_VEL
LIN {X 0,Y 295.495,Z 940.328,A -85,B 0,C 180,E1 16515.824,E2 16515.824} C_VEL
LIN {X 0,Y 323.469,Z 887.473,A -85,B 0,C 180,E1 16524.761,E2 16524.761} C_VEL
LIN {X 0,Y 346.518,Z 830.711,A -85,B 0,C 180,E1 16530.513,E2 16530.513} C_VEL
LIN {X 0,Y 341.838,Z 805.763,A -85,B 0,C 180,E1 16538.542,E2 16538.542} C_VEL
LIN {X 0,Y 339.743,Z 798.086,A -85,B 0,C 180,E1 16544.604,E2 16544.604} C_VEL
LIN {X 0,Y 336.85,Z 806.615,A -85,B 0,C 180,E1 16550.475,E2 16550.475} C_VEL
LIN {X 0,Y 338.524,Z 820.255,A -85,B 0,C 180,E1 16557.448,E2 16557.448} C_VEL
LIN {X 0,Y 338.797,Z 838.514,A -85,B 0,C 180,E1 16562.425,E2 16562.425} C_VEL
LIN {X 0,Y 310.957,Z 895.303,A -85,B 0,C 180,E1 16569.216,E2 16569.216} C_VEL
LIN {X 0,Y 283.35,Z 940.757,A -85,B 0,C 180,E1 16579.036,E2 16579.036} C_VEL
LIN {X 0,Y 262.567,Z 973.823,A -85,B 0,C 180,E1 16592.159,E2 16592.159} C_VEL
LIN {X 0,Y 253.045,Z 992.252,A -85,B 0,C 180,E1 16606.395,E2 16606.395} C_VEL
LIN {X 0,Y 250.017,Z 998.441,A -85,B 0,C 180,E1 16618.94,E2 16618.94} C_VEL
LIN {X 0,Y 251.463,Z 995.219,A -85,B 0,C 180,E1 16632.438,E2 16632.438} C_VEL
LIN {X 0,Y 257.821,Z 980.06,A -85,B 0,C 180,E1 16646.737,E2 16646.737} C_VEL
LIN {X 0,Y 274.761,Z 949.53,A -85,B 0,C 180,E1 16660.744,E2 16660.744} C_VEL
LIN {X 0,Y 299.05,Z 905.858,A -85,B 0,C 180,E1 16671.588,E2 16671.588} C_VEL
LIN {X 0,Y 324.839,Z 850.478,A -85,B 0,C 180,E1 16679.185,E2 16679.185} C_VEL
LIN {X 0,Y 330.807,Z 831.644,A -85,B 0,C 180,E1 16681.257,E2 16681.257} C_VEL
LIN {X 0,Y 320.143,Z 796.64,A -85,B 0,C 180,E1 16690.758,E2 16690.758} C_VEL
LIN {X 0,Y 307.131,Z 769.319,A -85,B 0,C 180,E1 16701.847,E2 16701.847} C_VEL
LIN {X 0,Y 298.048,Z 752.782,A -85,B 0,C 180,E1 16713.3,E2 16713.3} C_VEL
LIN {X 0,Y 295.048,Z 746.165,A -85,B 0,C 180,E1 16723.552,E2 16723.552} C_VEL
LIN {X 0,Y 297.05,Z 748.595,A -85,B 0,C 180,E1 16734.469,E2 16734.469} C_VEL
LIN {X 0,Y 304.595,Z 760.33,A -85,B 0,C 180,E1 16745.249,E2 16745.249} C_VEL
LIN {X 0,Y 317.588,Z 785.736,A -85,B 0,C 180,E1 16756.635,E2 16756.635} C_VEL
LIN {X 0,Y 331.059,Z 819.872,A -85,B 0,C 180,E1 16766.445,E2 16766.445} C_VEL
LIN {X 0,Y 334.418,Z 836.544,A -85,B 0,C 180,E1 16769.916,E2 16769.916} C_VEL
LIN {X 0,Y 309.626,Z 896.697,A -85,B 0,C 180,E1 16776.027,E2 16776.027} C_VEL
LIN {X 0,Y 284.572,Z 945.527,A -85,B 0,C 180,E1 16784.986,E2 16784.986} C_VEL
LIN {X 0,Y 264.516,Z 982.593,A -85,B 0,C 180,E1 16796.972,E2 16796.972} C_VEL
LIN {X 0,Y 252.98,Z 1007.52,A -85,B 0,C 180,E1 16812.081,E2 16812.081} C_VEL
LIN {X 0,Y 251.119,Z 1016.602,A -85,B 0,C 180,E1 16825.122,E2 16825.122} C_VEL
LIN {X 0,Y 251.202,Z 1016.547,A -85,B 0,C 180,E1 16835.199,E2 16835.199} C_VEL
LIN {X 0,Y 253.628,Z 1006.308,A -85,B 0,C 180,E1 16849.213,E2 16849.213} C_VEL
LIN {X 0,Y 264.892,Z 982.5,A -85,B 0,C 180,E1 16863.577,E2 16863.577} C_VEL
LIN {X 0,Y 287.466,Z 944.085,A -85,B 0,C 180,E1 16876.092,E2 16876.092} C_VEL
LIN {X 0,Y 315.377,Z 894.59,A -85,B 0,C 180,E1 16885.077,E2 16885.077} C_VEL
LIN {X 0,Y 341.571,Z 834.499,A -85,B 0,C 180,E1 16891.511,E2 16891.511} C_VEL
LIN {X 0,Y 338.061,Z 811.909,A -85,B 0,C 180,E1 16899.25,E2 16899.25} C_VEL
LIN {X 0,Y 336.428,Z 805.076,A -85,B 0,C 180,E1 16905.89,E2 16905.89} C_VEL
LIN {X 0,Y 336.85,Z 806.615,A -85,B 0,C 180,E1 16910.475,E2 16910.475} C_VEL
LIN {X 0,Y 334.195,Z 823.566,A -85,B 0,C 180,E1 16915.852,E2 16915.852} C_VEL
LIN {X 0,Y 333.592,Z 842.905,A -85,B 0,C 180,E1 16921.52,E2 16921.52} C_VEL
LIN {X 0,Y 305.014,Z 898.265,A -85,B 0,C 180,E1 16928.342,E2 16928.342} C_VEL
LIN {X 0,Y 275.139,Z 944.882,A -85,B 0,C 180,E1 16938.917,E2 16938.917} C_VEL
LIN {X 0,Y 253.365,Z 977.696,A -85,B 0,C 180,E1 16953.252,E2 16953.252} C_VEL
LIN {X 0,Y 244.811,Z 993.682,A -85,B 0,C 180,E1 16967.174,E2 16967.174} C_VEL
LIN {X 0,Y 241.851,Z 998.94,A -85,B 0,C 180,E1 16981.927,E2 16981.927} C_VEL
LIN {X 0,Y 244.495,Z 993.228,A -85,B 0,C 180,E1 16996.037,E2 16996.037} C_VEL
LIN {X 0,Y 254.109,Z 973.333,A -85,B 0,C 180,E1 17011.712,E2 17011.712} C_VEL
LIN {X 0,Y 274.367,Z 939.361,A -85,B 0,C 180,E1 17025.047,E2 17025.047} C_VEL
LIN {X 0,Y 300.547,Z 892.714,A -85,B 0,C 180,E1 17035.018,E2 17035.018} C_VEL
LIN {X 0,Y 325.315,Z 836.41,A -85,B 0,C 180,E1 17041.846,E2 17041.846} C_VEL
LIN {X 0,Y 315.822,Z 802.859,A -85,B 0,C 180,E1 17051.222,E2 17051.222} C_VEL
LIN {X 0,Y 304.105,Z 776.63,A -85,B 0,C 180,E1 17062.092,E2 17062.092} C_VEL
LIN {X 0,Y 295.621,Z 760.215,A -85,B 0,C 180,E1 17073.796,E2 17073.796} C_VEL
LIN {X 0,Y 293.106,Z 753.93,A -85,B 0,C 180,E1 17083.44,E2 17083.44} C_VEL
LIN {X 0,Y 295.016,Z 756.311,A -85,B 0,C 180,E1 17094.347,E2 17094.347} C_VEL
LIN {X 0,Y 301.952,Z 767.756,A -85,B 0,C 180,E1 17104.934,E2 17104.934} C_VEL
LIN {X 0,Y 314.64,Z 793.861,A -85,B 0,C 180,E1 17116.708,E2 17116.708} C_VEL
LIN {X 0,Y 327.031,Z 828.384,A -85,B 0,C 180,E1 17126.679,E2 17126.679} C_VEL
LIN {X 0,Y 328.308,Z 840.722,A -85,B 0,C 180,E1 17129.089,E2 17129.089} C_VEL
LIN {X 0,Y 303.142,Z 899.33,A -85,B 0,C 180,E1 17135.242,E2 17135.242} C_VEL
LIN {X 0,Y 276.01,Z 949.592,A -85,B 0,C 180,E1 17144.934,E2 17144.934} C_VEL
LIN {X 0,Y 255.359,Z 985.786,A -85,B 0,C 180,E1 17157.664,E2 17157.664} C_VEL
LIN {X 0,Y 245.028,Z 1007.661,A -85,B 0,C 180,E1 17171.959,E2 17171.959} C_VEL
LIN {X 0,Y 243.107,Z 1016.19,A -85,B 0,C 180,E1 17184.626,E2 17184.626} C_VEL
LIN {X 0,Y 243.19,Z 1016.255,A -85,B 0,C 180,E1 17195.37,E2 17195.37} C_VEL
LIN {X 0,Y 245.827,Z 1006.049,A -85,B 0,C 180,E1 17209.848,E2 17209.848} C_VEL
LIN {X 0,Y 257.942,Z 982.311,A -85,B 0,C 180,E1 17224.608,E2 17224.608} C_VEL
LIN {X 0,Y 282.257,Z 943.299,A -85,B 0,C 180,E1 17237.51,E2 17237.51} C_VEL
LIN {X 0,Y 311.85,Z 893.021,A -85,B 0,C 180,E1 17246.562,E2 17246.562} C_VEL
LIN {X 0,Y 336.769,Z 839.741,A -85,B 0,C 180,E1 17252.137,E2 17252.137} C_VEL
LIN {X 0,Y 334.542,Z 819.438,A -85,B 0,C 180,E1 17259.217,E2 17259.217} C_VEL
LIN {X 0,Y 333.165,Z 812.502,A -85,B 0,C 180,E1 17265.515,E2 17265.515} C_VEL
LIN {X 0,Y 333.814,Z 816.712,A -85,B 0,C 180,E1 17272.664,E2 17272.664} C_VEL
LIN {X 0,Y 334.195,Z 823.566,A -85,B 0,C 180,E1 17275.852,E2 17275.852} C_VEL
LIN {X 0,Y 329.898,Z 839.744,A -85,B 0,C 180,E1 17278.819,E2 17278.819} C_VEL
LIN {X 0,Y 327.747,Z 849.044,A -85,B 0,C 180,E1 17280.748,E2 17280.748} C_VEL
LIN {X 0,Y 297.77,Z 903.341,A -85,B 0,C 180,E1 17287.82,E2 17287.82} C_VEL
LIN {X 0,Y 268.252,Z 946.795,A -85,B 0,C 180,E1 17298.145,E2 17298.145} C_VEL
LIN {X 0,Y 245.719,Z 978.913,A -85,B 0,C 180,E1 17312.809,E2 17312.809} C_VEL
LIN {X 0,Y 236.633,Z 994.703,A -85,B 0,C 180,E1 17327.672,E2 17327.672} C_VEL
LIN {X 0,Y 233.826,Z 999.25,A -85,B 0,C 180,E1 17341.201,E2 17341.201} C_VEL
LIN {X 0,Y 236.377,Z 994.088,A -85,B 0,C 180,E1 17355.653,E2 17355.653} C_VEL
LIN {X 0,Y 246.052,Z 975.001,A -85,B 0,C 180,E1 17371.768,E2 17371.768} C_VEL
LIN {X 0,Y 266.403,Z 942.577,A -85,B 0,C 180,E1 17385.295,E2 17385.295} C_VEL
LIN {X 0,Y 293.494,Z 896.444,A -85,B 0,C 180,E1 17395.662,E2 17395.662} C_VEL
LIN {X 0,Y 319.54,Z 839.745,A -85,B 0,C 180,E1 17402.779,E2 17402.779} C_VEL
LIN {X 0,Y 310.864,Z 807.287,A -85,B 0,C 180,E1 17412.313,E2 17412.313} C_VEL
LIN {X 0,Y 300.045,Z 781.402,A -85,B 0,C 180,E1 17423.572,E2 17423.572} C_VEL
LIN {X 0,Y 292.411,Z 766.958,A -85,B 0,C 180,E1 17435.454,E2 17435.454} C_VEL
LIN {X 0,Y 290.922,Z 761.564,A -85,B 0,C 180,E1 17444.81,E2 17444.81} C_VEL
LIN {X 0,Y 292.803,Z 764.187,A -85,B 0,C 180,E1 17454.312,E2 17454.312} C_VEL
LIN {X 0,Y 299.049,Z 774.676,A -85,B 0,C 180,E1 17464.344,E2 17464.344} C_VEL
LIN {X 0,Y 310.989,Z 800.927,A -85,B 0,C 180,E1 17476.454,E2 17476.454} C_VEL
LIN {X 0,Y 322.389,Z 835.367,A -85,B 0,C 180,E1 17486.533,E2 17486.533} C_VEL
LIN {X 0,Y 322.756,Z 843.633,A -85,B 0,C 180,E1 17488.137,E2 17488.137} C_VEL
LIN {X 0,Y 297.429,Z 900.195,A -85,B 0,C 180,E1 17494.186,E2 17494.186} C_VEL
LIN {X 0,Y 269.248,Z 950.438,A -85,B 0,C 180,E1 17504.057,E2 17504.057} C_VEL
LIN {X 0,Y 247.249,Z 987.112,A -85,B 0,C 180,E1 17517.515,E2 17517.515} C_VEL
LIN {X 0,Y 236.558,Z 1009.078,A -85,B 0,C 180,E1 17533.22,E2 17533.22} C_VEL
LIN {X 0,Y 235.129,Z 1015.872,A -85,B 0,C 180,E1 17544.443,E2 17544.443} C_VEL
LIN {X 0,Y 235.19,Z 1015.967,A -85,B 0,C 180,E1 17555.554,E2 17555.554} C_VEL
LIN {X 0,Y 238.043,Z 1005.796,A -85,B 0,C 180,E1 17570.526,E2 17570.526} C_VEL
LIN {X 0,Y 251.456,Z 981.636,A -85,B 0,C 180,E1 17585.937,E2 17585.937} C_VEL
LIN {X 0,Y 277.73,Z 941.892,A -85,B 0,C 180,E1 17599.129,E2 17599.129} C_VEL
LIN {X 0,Y 308.464,Z 891.676,A -85,B 0,C 180,E1 17608.066,E2 17608.066} C_VEL
LIN {X 0,Y 331.972,Z 844.017,A -85,B 0,C 180,E1 17613.053,E2 17613.053} C_VEL
LIN {X 0,Y 330.482,Z 824.906,A -85,B 0,C 180,E1 17620.281,E2 17620.281} C_VEL
LIN {X 0,Y 329.721,Z 819.598,A -85,B 0,C 180,E1 17628.069,E2 17628.069} C_VEL
LIN {X 0,Y 330.083,Z 828.353,A -85,B 0,C 180,E1 17634.744,E2 17634.744} C_VEL
LIN {X 0,Y 329.898,Z 839.744,A -85,B 0,C 180,E1 17638.819,E2 17638.819} C_VEL
LIN {X 0,Y 325.925,Z 848.825,A -85,B 0,C 180,E1 17639.828,E2 17639.828} C_VEL
LIN {X 0,Y 319.593,Z 859.444,A -85,B 0,C 180,E1 17640.414,E2 17640.414} C_VEL
LIN {X 0,Y 287.692,Z 912.62,A -85,B 0,C 180,E1 17648.09,E2 17648.09} C_VEL
LIN {X 0,Y 256.837,Z 954.903,A -85,B 0,C 180,E1 17659.557,E2 17659.557} C_VEL
LIN {X 0,Y 235.566,Z 983.961,A -85,B 0,C 180,E1 17675.222,E2 17675.222} C_VEL
LIN {X 0,Y 227.688,Z 997.051,A -85,B 0,C 180,E1 17690.715,E2 17690.715} C_VEL
LIN {X 0,Y 225.961,Z 999.209,A -85,B 0,C 180,E1 17705.069,E2 17705.069} C_VEL
LIN {X 0,Y 229.328,Z 992.446,A -85,B 0,C 180,E1 17718.55,E2 17718.55} C_VEL
LIN {X 0,Y 240.701,Z 972.154,A -85,B 0,C 180,E1 17734.521,E2 17734.521} C_VEL
LIN {X 0,Y 264.25,Z 936.336,A -85,B 0,C 180,E1 17748.414,E2 17748.414} C_VEL
LIN {X 0,Y 292.942,Z 888.275,A -85,B 0,C 180,E1 17758.199,E2 17758.199} C_VEL
LIN {X 0,Y 313.735,Z 842.9,A -85,B 0,C 180,E1 17763.799,E2 17763.799} C_VEL
LIN {X 0,Y 305.859,Z 811.543,A -85,B 0,C 180,E1 17773.487,E2 17773.487} C_VEL
LIN {X 0,Y 296.335,Z 787.545,A -85,B 0,C 180,E1 17784.495,E2 17784.495} C_VEL
LIN {X 0,Y 290.877,Z 775.589,A -85,B 0,C 180,E1 17793.662,E2 17793.662} C_VEL
LIN {X 0,Y 288.747,Z 769.319,A -85,B 0,C 180,E1 17803.183,E2 17803.183} C_VEL
LIN {X 0,Y 290.369,Z 771.615,A -85,B 0,C 180,E1 17813.982,E2 17813.982} C_VEL
LIN {X 0,Y 296.95,Z 784.364,A -85,B 0,C 180,E1 17825.312,E2 17825.312} C_VEL
LIN {X 0,Y 308.167,Z 810.366,A -85,B 0,C 180,E1 17837.07,E2 17837.07} C_VEL
LIN {X 0,Y 317.945,Z 844.283,A -85,B 0,C 180,E1 17846.934,E2 17846.934} C_VEL
LIN {X 0,Y 291.249,Z 902.088,A -85,B 0,C 180,E1 17853.242,E2 17853.242} C_VEL
LIN {X 0,Y 262.541,Z 951.205,A -85,B 0,C 180,E1 17863.132,E2 17863.132} C_VEL
LIN {X 0,Y 239.143,Z 988.433,A -85,B 0,C 180,E1 17877.356,E2 17877.356} C_VEL
LIN {X 0,Y 228.742,Z 1008.709,A -85,B 0,C 180,E1 17892.628,E2 17892.628} C_VEL
LIN {X 0,Y 227.12,Z 1015.553,A -85,B 0,C 180,E1 17904.247,E2 17904.247} C_VEL
LIN {X 0,Y 227.177,Z 1015.679,A -85,B 0,C 180,E1 17915.75,E2 17915.75} C_VEL
LIN {X 0,Y 230.309,Z 1005.556,A -85,B 0,C 180,E1 17931.248,E2 17931.248} C_VEL
LIN {X 0,Y 244.883,Z 981.317,A -85,B 0,C 180,E1 17947.172,E2 17947.172} C_VEL
LIN {X 0,Y 273.105,Z 940.983,A -85,B 0,C 180,E1 17960.696,E2 17960.696} C_VEL
LIN {X 0,Y 305.537,Z 890.02,A -85,B 0,C 180,E1 17969.655,E2 17969.655} C_VEL
LIN {X 0,Y 327.181,Z 847.247,A -85,B 0,C 180,E1 17974.309,E2 17974.309} C_VEL
LIN {X 0,Y 326.549,Z 830.482,A -85,B 0,C 180,E1 17981.363,E2 17981.363} C_VEL
LIN {X 0,Y 326.091,Z 826.74,A -85,B 0,C 180,E1 17987.934,E2 17987.934} C_VEL
LIN {X 0,Y 325.871,Z 835.546,A -85,B 0,C 180,E1 17994.676,E2 17994.676} C_VEL
LIN {X 0,Y 323.765,Z 851.418,A -85,B 0,C 180,E1 17999.599,E2 17999.599} C_VEL
LIN {X 0,Y 319.593,Z 859.444,A -85,B 0,C 180,E1 18000.414,E2 18000.414} C_VEL
LIN {X 0,Y 300.592,Z 887.455,A -85,B 0,C 180,E1 18002.382,E2 18002.382} C_VEL
LIN {X 0,Y 266.335,Z 936.072,A -85,B 0,C 180,E1 18011.955,E2 18011.955} C_VEL
LIN {X 0,Y 238.22,Z 971.305,A -85,B 0,C 180,E1 18025.578,E2 18025.578} C_VEL
LIN {X 0,Y 222.784,Z 992.16,A -85,B 0,C 180,E1 18041.939,E2 18041.939} C_VEL
LIN {X 0,Y 218.693,Z 998.777,A -85,B 0,C 180,E1 18053.855,E2 18053.855} C_VEL
LIN {X 0,Y 218.535,Z 998.253,A -85,B 0,C 180,E1 18069.657,E2 18069.657} C_VEL
LIN {X 0,Y 224.265,Z 987.084,A -85,B 0,C 180,E1 18085.149,E2 18085.149} C_VEL
LIN {X 0,Y 241.021,Z 961.557,A -85,B 0,C 180,E1 18100.889,E2 18100.889} C_VEL
LIN {X 0,Y 267.99,Z 921.86,A -85,B 0,C 180,E1 18113.354,E2 18113.354} C_VEL
LIN {X 0,Y 297.059,Z 871.51,A -85,B 0,C 180,E1 18121.793,E2 18121.793} C_VEL
LIN {X 0,Y 308.024,Z 846.162,A -85,B 0,C 180,E1 18124.833,E2 18124.833} C_VEL
LIN {X 0,Y 300.808,Z 815.752,A -85,B 0,C 180,E1 18134.706,E2 18134.706} C_VEL
LIN {X 0,Y 292.428,Z 793.67,A -85,B 0,C 180,E1 18145.509,E2 18145.509} C_VEL
LIN {X 0,Y 286.894,Z 781.486,A -85,B 0,C 180,E1 18156.612,E2 18156.612} C_VEL
LIN {X 0,Y 286.243,Z 776.768,A -85,B 0,C 180,E1 18166.181,E2 18166.181} C_VEL
LIN {X 0,Y 287.933,Z 779.631,A -85,B 0,C 180,E1 18174.356,E2 18174.356} C_VEL
LIN {X 0,Y 294.139,Z 792.179,A -85,B 0,C 180,E1 18185.363,E2 18185.363} C_VEL
LIN {X 0,Y 304.022,Z 816.821,A -85,B 0,C 180,E1 18196.653,E2 18196.653} C_VEL
LIN {X 0,Y 312.322,Z 847.859,A -85,B 0,C 180,E1 18205.981,E2 18205.981} C_VEL
LIN {X 0,Y 284.065,Z 905.925,A -85,B 0,C 180,E1 18212.563,E2 18212.563} C_VEL
LIN {X 0,Y 254.862,Z 953.429,A -85,B 0,C 180,E1 18222.597,E2 18222.597} C_VEL
LIN {X 0,Y 231.341,Z 989.143,A -85,B 0,C 180,E1 18236.935,E2 18236.935} C_VEL
